LIN {X 0,Y 314.358,Z 529.66,A -85,B 0,C 180,E1 14023.753,E2 14023.753} C_VEL
LIN {X 0,Y 314.841,Z 529.66,A -85,B 0,C 180,E1 14031.737,E2 14031.737} C_VEL
LIN {X 0,Y 315.373,Z 529.66,A -85,B 0,C 180,E1 14037.261,E2 14037.261} C_VEL
LIN {X 0,Y 315.324,Z 529.66,A -85,B 0,C 180,E1 14042.747,E2 14042.747} C_VEL
LIN {X 0,Y 314.746,Z 529.66,A -85,B 0,C 180,E1 14051.06,E2 14051.06} C_VEL
LIN {X 0,Y 314.38,Z 529.66,A -85,B 0,C 180,E1 14056.741,E2 14056.741} C_VEL
LIN {X 0,Y 313.895,Z 529.66,A -85,B 0,C 180,E1 14064.019,E2 14064.019} C_VEL
LIN {X 0,Y 313.702,Z 529.66,A -85,B 0,C 180,E1 14072.529,E2 14072.529} C_VEL
LIN {X 0,Y 331.392,Z 572.539,A -85,B 0,C 180,E1 14075.795,E2 14075.795} C_VEL
LIN {X 0,Y 335.77,Z 585.842,A -85,B 0,C 180,E1 14076.583,E2 14076.583} C_VEL
LIN {X 0,Y 334.083,Z 636.564,A -85,B 0,C 180,E1 14077.88,E2 14077.88} C_VEL
LIN {X 0,Y 331.433,Z 665.303,A -85,B 0,C 180,E1 14079.603,E2 14079.603} C_VEL
LIN {X 0,Y 327.822,Z 690.981,A -85,B 0,C 180,E1 14082.214,E2 14082.214} C_VEL
LIN {X 0,Y 323.741,Z 713,A -85,B 0,C 180,E1 14085.638,E2 14085.638} C_VEL
LIN {X 0,Y 320.247,Z 730.569,A -85,B 0,C 180,E1 14089.741,E2 14089.741} C_VEL
LIN {X 0,Y 317.778,Z 743.68,A -85,B 0,C 180,E1 14094.497,E2 14094.497} C_VEL
LIN {X 0,Y 316.381,Z 751.07,A -85,B 0,C 180,E1 14099.156,E2 14099.156} C_VEL
LIN {X 0,Y 315.419,Z 754.016,A -85,B 0,C 180,E1 14104.495,E2 14104.495} C_VEL
LIN {X 0,Y 315.966,Z 751.687,A -85,B 0,C 180,E1 14109.434,E2 14109.434} C_VEL
LIN {X 0,Y 317.161,Z 744.828,A -85,B 0,C 180,E1 14114.122,E2 14114.122} C_VEL
LIN {X 0,Y 319.364,Z 731.71,A -85,B 0,C 180,E1 14119.104,E2 14119.104} C_VEL
LIN {X 0,Y 322.445,Z 714.366,A -85,B 0,C 180,E1 14123.28,E2 14123.28} C_VEL
LIN {X 0,Y 326.093,Z 692.368,A -85,B 0,C 180,E1 14126.826,E2 14126.826} C_VEL
LIN {X 0,Y 329.646,Z 666.051,A -85,B 0,C 180,E1 14129.589,E2 14129.589} C_VEL
LIN {X 0,Y 332.227,Z 637.274,A -85,B 0,C 180,E1 14131.367,E2 14131.367} C_VEL
LIN {X 0,Y 333.756,Z 589.127,A -85,B 0,C 180,E1 14132.637,E2 14132.637} C_VEL
LIN {X 0,Y 332.654,Z 578.727,A -85,B 0,C 180,E1 14132.982,E2 14132.982} C_VEL
LIN {X 0,Y 319.042,Z 540.423,A -85,B 0,C 180,E1 14135.188,E2 14135.188} C_VEL
LIN {X 0,Y 314.996,Z 529.66,A -85,B 0,C 180,E1 14136.014,E2 14136.014} C_VEL
LIN {X 0,Y 314.466,Z 529.66,A -85,B 0,C 180,E1 14143.881,E2 14143.881} C_VEL
LIN {X 0,Y 314.137,Z 529.66,A -85,B 0,C 180,E1 14149.647,E2 14149.647} C_VEL
LIN {X 0,Y 313.832,Z 529.66,A -85,B 0,C 180,E1 14155.641,E2 14155.641} C_VEL
LIN {X 0,Y 313.606,Z 529.66,A -85,B 0,C 180,E1 14161.956,E2 14161.956} C_VEL
LIN {X 0,Y 313.395,Z 529.66,A -85,B 0,C 180,E1 14169.605,E2 14169.605} C_VEL
LIN {X 0,Y 313.39,Z 529.66,A -85,B 0,C 180,E1 14177.611,E2 14177.611} C_VEL
LIN {X 0,Y 313.516,Z 529.661,A -85,B 0,C 180,E1 14178.724,E2 14178.724} C_VEL
LIN {X 0,Y 333.561,Z 579.091,A -85,B 0,C 180,E1 14182.875,E2 14182.875} C_VEL
LIN {X 0,Y 341.105,Z 602.01,A -85,B 0,C 180,E1 14185.002,E2 14185.002} C_VEL
LIN {X 0,Y 335.859,Z 636.992,A -85,B 0,C 180,E1 14187.695,E2 14187.695} C_VEL
LIN {X 0,Y 330.121,Z 668.653,A -85,B 0,C 180,E1 14191.314,E2 14191.314} C_VEL
LIN {X 0,Y 324.858,Z 695.392,A -85,B 0,C 180,E1 14195.65,E2 14195.65} C_VEL
LIN {X 0,Y 320.51,Z 717.686,A -85,B 0,C 180,E1 14200.754,E2 14200.754} C_VEL
LIN {X 0,Y 317.677,Z 734.305,A -85,B 0,C 180,E1 14206.257,E2 14206.257} C_VEL
LIN {X 0,Y 316.286,Z 745.604,A -85,B 0,C 180,E1 14212.1,E2 14212.1} C_VEL
LIN {X 0,Y 315.85,Z 751.035,A -85,B 0,C 180,E1 14217.258,E2 14217.258} C_VEL
LIN {X 0,Y 316.055,Z 752.334,A -85,B 0,C 180,E1 14222.733,E2 14222.733} C_VEL
LIN {X 0,Y 316.668,Z 749.149,A -85,B 0,C 180,E1 14228.215,E2 14228.215} C_VEL
LIN {X 0,Y 318.78,Z 740.37,A -85,B 0,C 180,E1 14234.24,E2 14234.24} C_VEL
LIN {X 0,Y 322.751,Z 725.649,A -85,B 0,C 180,E1 14240.202,E2 14240.202} C_VEL
LIN {X 0,Y 329.291,Z 704.647,A -85,B 0,C 180,E1 14245.803,E2 14245.803} C_VEL
LIN {X 0,Y 337.651,Z 677.968,A -85,B 0,C 180,E1 14250.736,E2 14250.736} C_VEL
LIN {X 0,Y 347.649,Z 645.626,A -85,B 0,C 180,E1 14254.914,E2 14254.914} C_VEL
LIN {X 0,Y 358.765,Z 606.435,A -85,B 0,C 180,E1 14258.535,E2 14258.535} C_VEL
LIN {X 0,Y 359.21,Z 596.015,A -85,B 0,C 180,E1 14260.875,E2 14260.875} C_VEL
LIN {X 0,Y 359.26,Z 593.944,A -85,B 0,C 180,E1 14262.22,E2 14262.22} C_VEL
LIN {X 0,Y 359.589,Z 594.189,A -85,B 0,C 180,E1 14263.651,E2 14263.651} C_VEL
LIN {X 0,Y 359.874,Z 599.525,A -85,B 0,C 180,E1 14265.46,E2 14265.46} C_VEL
LIN {X 0,Y 359.344,Z 611.481,A -85,B 0,C 180,E1 14267.298,E2 14267.298} C_VEL
LIN {X 0,Y 348.056,Z 653.394,A -85,B 0,C 180,E1 14270.652,E2 14270.652} C_VEL
LIN {X 0,Y 338.01,Z 689.08,A -85,B 0,C 180,E1 14274.803,E2 14274.803} C_VEL
LIN {X 0,Y 329.433,Z 719.409,A -85,B 0,C 180,E1 14279.745,E2 14279.745} C_VEL
LIN {X 0,Y 322.989,Z 743.295,A -85,B 0,C 180,E1 14285.137,E2 14285.137} C_VEL
LIN {X 0,Y 318.517,Z 762.82,A -85,B 0,C 180,E1 14291.34,E2 14291.34} C_VEL
LIN {X 0,Y 316.479,Z 775.559,A -85,B 0,C 180,E1 14297.373,E2 14297.373} C_VEL
LIN {X 0,Y 315.859,Z 782.903,A -85,B 0,C 180,E1 14303.142,E2 14303.142} C_VEL
LIN {X 0,Y 315.765,Z 785.334,A -85,B 0,C 180,E1 14307.262,E2 14307.262} C_VEL
LIN {X 0,Y 315.855,Z 784.953,A -85,B 0,C 180,E1 14312.74,E2 14312.74} C_VEL
LIN {X 0,Y 315.941,Z 780.256,A -85,B 0,C 180,E1 14318.239,E2 14318.239} C_VEL
LIN {X 0,Y 316.897,Z 769.663,A -85,B 0,C 180,E1 14324.478,E2 14324.478} C_VEL
LIN {X 0,Y 319.276,Z 753.654,A -85,B 0,C 180,E1 14330.401,E2 14330.401} C_VEL
LIN {X 0,Y 323.428,Z 732.194,A -85,B 0,C 180,E1 14335.939,E2 14335.939} C_VEL
LIN {X 0,Y 325.518,Z 722.568,A -85,B 0,C 180,E1 14337.919,E2 14337.919} C_VEL
LIN {X 0,Y 324.253,Z 710.874,A -85,B 0,C 180,E1 14340.211,E2 14340.211} C_VEL
LIN {X 0,Y 323.099,Z 698.429,A -85,B 0,C 180,E1 14342.396,E2 14342.396} C_VEL
LIN {X 0,Y 329.898,Z 665.459,A -85,B 0,C 180,E1 14346.488,E2 14346.488} C_VEL
LIN {X 0,Y 336.27,Z 629.393,A -85,B 0,C 180,E1 14349.577,E2 14349.577} C_VEL
LIN {X 0,Y 338.64,Z 610.74,A -85,B 0,C 180,E1 14350.76,E2 14350.76} C_VEL
LIN {X 0,Y 324.137,Z 572.197,A -85,B 0,C 180,E1 14354.249,E2 14354.249} C_VEL
LIN {X 0,Y 305.579,Z 529.66,A -85,B 0,C 180,E1 14358.2,E2 14358.2} C_VEL
LIN {X 0,Y 305.614,Z 529.66,A -85,B 0,C 180,E1 14367.108,E2 14367.108} C_VEL
LIN {X 0,Y 305.857,Z 529.66,A -85,B 0,C 180,E1 14373.643,E2 14373.643} C_VEL
LIN {X 0,Y 306.152,Z 529.66,A -85,B 0,C 180,E1 14379.821,E2 14379.821} C_VEL
LIN {X 0,Y 306.519,Z 529.66,A -85,B 0,C 180,E1 14385.754,E2 14385.754} C_VEL
LIN {X 0,Y 306.894,Z 529.66,A -85,B 0,C 180,E1 14391.521,E2 14391.521} C_VEL
LIN {X 0,Y 307.45,Z 529.66,A -85,B 0,C 180,E1 14397.191,E2 14397.191} C_VEL
LIN {X 0,Y 307.404,Z 529.66,A -85,B 0,C 180,E1 14402.817,E2 14402.817} C_VEL
LIN {X 0,Y 306.811,Z 529.66,A -85,B 0,C 180,E1 14411.35,E2 14411.35} C_VEL
LIN {X 0,Y 306.396,Z 529.66,A -85,B 0,C 180,E1 14417.191,E2 14417.191} C_VEL
LIN {X 0,Y 306.041,Z 529.66,A -85,B 0,C 180,E1 14423.236,E2 14423.236} C_VEL
LIN {X 0,Y 305.753,Z 529.66,A -85,B 0,C 180,E1 14431.48,E2 14431.48} C_VEL
LIN {X 0,Y 323.99,Z 572.634,A -85,B 0,C 180,E1 14434.995,E2 14434.995} C_VEL
LIN {X 0,Y 328.959,Z 588.44,A -85,B 0,C 180,E1 14435.949,E2 14435.949} C_VEL
LIN {X 0,Y 327.127,Z 637.889,A -85,B 0,C 180,E1 14437.26,E2 14437.26} C_VEL
LIN {X 0,Y 324.455,Z 665.524,A -85,B 0,C 180,E1 14438.961,E2 14438.961} C_VEL
LIN {X 0,Y 320.62,Z 691.541,A -85,B 0,C 180,E1 14441.656,E2 14441.656} C_VEL
LIN {X 0,Y 316.272,Z 713.758,A -85,B 0,C 180,E1 14445.199,E2 14445.199} C_VEL
LIN {X 0,Y 312.4,Z 732.228,A -85,B 0,C 180,E1 14449.7,E2 14449.7} C_VEL
LIN {X 0,Y 309.987,Z 744.201,A -85,B 0,C 180,E1 14454.256,E2 14454.256} C_VEL
LIN {X 0,Y 308.375,Z 752.077,A -85,B 0,C 180,E1 14459.556,E2 14459.556} C_VEL
LIN {X 0,Y 307.546,Z 754.341,A -85,B 0,C 180,E1 14463.793,E2 14463.793} C_VEL
LIN {X 0,Y 307.872,Z 752.827,A -85,B 0,C 180,E1 14468.64,E2 14468.64} C_VEL
LIN {X 0,Y 309.126,Z 746.371,A -85,B 0,C 180,E1 14473.698,E2 14473.698} C_VEL
LIN {X 0,Y 311.331,Z 733.969,A -85,B 0,C 180,E1 14478.82,E2 14478.82} C_VEL
LIN {X 0,Y 314.366,Z 717.563,A -85,B 0,C 180,E1 14483.107,E2 14483.107} C_VEL
LIN {X 0,Y 318.132,Z 696.355,A -85,B 0,C 180,E1 14486.818,E2 14486.818} C_VEL
LIN {X 0,Y 321.802,Z 671.686,A -85,B 0,C 180,E1 14489.663,E2 14489.663} C_VEL
LIN {X 0,Y 324.629,Z 643.608,A -85,B 0,C 180,E1 14491.662,E2 14491.662} C_VEL
LIN {X 0,Y 326.15,Z 611.366,A -85,B 0,C 180,E1 14492.747,E2 14492.747} C_VEL
LIN {X 0,Y 326.263,Z 582.825,A -85,B 0,C 180,E1 14493.443,E2 14493.443} C_VEL
LIN {X 0,Y 312.895,Z 544.522,A -85,B 0,C 180,E1 14495.694,E2 14495.694} C_VEL
LIN {X 0,Y 307.04,Z 529.66,A -85,B 0,C 180,E1 14496.791,E2 14496.791} C_VEL
LIN {X 0,Y 306.534,Z 529.66,A -85,B 0,C 180,E1 14504.248,E2 14504.248} C_VEL
LIN {X 0,Y 306.028,Z 529.66,A -85,B 0,C 180,E1 14513.232,E2 14513.232} C_VEL
LIN {X 0,Y 305.731,Z 529.66,A -85,B 0,C 180,E1 14519.574,E2 14519.574} C_VEL
LIN {X 0,Y 305.424,Z 529.66,A -85,B 0,C 180,E1 14527.762,E2 14527.762} C_VEL
LIN {X 0,Y 305.501,Z 529.66,A -85,B 0,C 180,E1 14533.748,E2 14533.748} C_VEL
LIN {X 0,Y 305.523,Z 529.888,A -85,B 0,C 180,E1 14537.803,E2 14537.803} C_VEL
LIN {X 0,Y 325.664,Z 578.93,A -85,B 0,C 180,E1 14542.105,E2 14542.105} C_VEL
LIN {X 0,Y 333.718,Z 604.557,A -85,B 0,C 180,E1 14544.541,E2 14544.541} C_VEL
LIN {X 0,Y 328.331,Z 638.995,A -85,B 0,C 180,E1 14547.311,E2 14547.311} C_VEL
LIN {X 0,Y 322.326,Z 670.994,A -85,B 0,C 180,E1 14551.129,E2 14551.129} C_VEL
LIN {X 0,Y 316.772,Z 698.028,A -85,B 0,C 180,E1 14555.737,E2 14555.737} C_VEL
LIN {X 0,Y 312.44,Z 719.749,A -85,B 0,C 180,E1 14560.97,E2 14560.97} C_VEL
LIN {X 0,Y 309.608,Z 736.118,A -85,B 0,C 180,E1 14566.718,E2 14566.718} C_VEL
LIN {X 0,Y 308.409,Z 745.967,A -85,B 0,C 180,E1 14572.065,E2 14572.065} C_VEL
LIN {X 0,Y 307.959,Z 751.348,A -85,B 0,C 180,E1 14577.188,E2 14577.188} C_VEL
LIN {X 0,Y 308.171,Z 752.848,A -85,B 0,C 180,E1 14582.803,E2 14582.803} C_VEL
LIN {X 0,Y 308.884,Z 749.882,A -85,B 0,C 180,E1 14588.424,E2 14588.424} C_VEL
LIN {X 0,Y 311.217,Z 741.069,A -85,B 0,C 180,E1 14594.743,E2 14594.743} C_VEL
LIN {X 0,Y 315.609,Z 726.484,A -85,B 0,C 180,E1 14600.863,E2 14600.863} C_VEL
LIN {X 0,Y 322.412,Z 706.547,A -85,B 0,C 180,E1 14606.395,E2 14606.395} C_VEL
LIN {X 0,Y 331.615,Z 679.844,A -85,B 0,C 180,E1 14611.549,E2 14611.549} C_VEL
LIN {X 0,Y 342.737,Z 647.661,A -85,B 0,C 180,E1 14615.877,E2 14615.877} C_VEL
LIN {X 0,Y 354.943,Z 610.837,A -85,B 0,C 180,E1 14619.396,E2 14619.396} C_VEL
LIN {X 0,Y 356.118,Z 602.755,A -85,B 0,C 180,E1 14621.307,E2 14621.307} C_VEL
LIN {X 0,Y 356.354,Z 601.212,A -85,B 0,C 180,E1 14622.645,E2 14622.645} C_VEL
LIN {X 0,Y 356.581,Z 602.503,A -85,B 0,C 180,E1 14623.996,E2 14623.996} C_VEL
LIN {X 0,Y 355.793,Z 610.922,A -85,B 0,C 180,E1 14625.831,E2 14625.831} C_VEL
LIN {X 0,Y 353.664,Z 619.82,A -85,B 0,C 180,E1 14626.696,E2 14626.696} C_VEL
LIN {X 0,Y 341.465,Z 659.253,A -85,B 0,C 180,E1 14630.151,E2 14630.151} C_VEL
LIN {X 0,Y 330.11,Z 695.501,A -85,B 0,C 180,E1 14634.755,E2 14634.755} C_VEL
LIN {X 0,Y 321.145,Z 724.9,A -85,B 0,C 180,E1 14640.03,E2 14640.03} C_VEL
LIN {X 0,Y 314.432,Z 748.303,A -85,B 0,C 180,E1 14645.916,E2 14645.916} C_VEL
LIN {X 0,Y 310.069,Z 766.678,A -85,B 0,C 180,E1 14652.533,E2 14652.533} C_VEL
LIN {X 0,Y 308.382,Z 777.819,A -85,B 0,C 180,E1 14658.714,E2 14658.714} C_VEL
LIN {X 0,Y 307.923,Z 783.588,A -85,B 0,C 180,E1 14664.377,E2 14664.377} C_VEL
LIN {X 0,Y 308.005,Z 785.155,A -85,B 0,C 180,E1 14670.001,E2 14670.001} C_VEL
LIN {X 0,Y 307.938,Z 782.501,A -85,B 0,C 180,E1 14675.626,E2 14675.626} C_VEL
LIN {X 0,Y 308.489,Z 774.306,A -85,B 0,C 180,E1 14681.976,E2 14681.976} C_VEL
LIN {X 0,Y 310.305,Z 760.118,A -85,B 0,C 180,E1 14688.366,E2 14688.366} C_VEL
LIN {X 0,Y 313.903,Z 740.758,A -85,B 0,C 180,E1 14694.194,E2 14694.194} C_VEL
LIN {X 0,Y 319.199,Z 716.347,A -85,B 0,C 180,E1 14699.442,E2 14699.442} C_VEL
LIN {X 0,Y 323.099,Z 698.429,A -85,B 0,C 180,E1 14702.396,E2 14702.396} C_VEL
LIN {X 0,Y 322.145,Z 685.268,A -85,B 0,C 180,E1 14704.454,E2 14704.454} C_VEL
LIN {X 0,Y 321.126,Z 673.313,A -85,B 0,C 180,E1 14706.165,E2 14706.165} C_VEL
LIN {X 0,Y 321.449,Z 671.49,A -85,B 0,C 180,E1 14706.381,E2 14706.381} C_VEL
LIN {X 0,Y 328.131,Z 636.403,A -85,B 0,C 180,E1 14709.66,E2 14709.66} C_VEL
LIN {X 0,Y 331.334,Z 612.5,A -85,B 0,C 180,E1 14711.302,E2 14711.302} C_VEL
LIN {X 0,Y 317.076,Z 574.226,A -85,B 0,C 180,E1 14714.919,E2 14714.919} C_VEL
LIN {X 0,Y 297.595,Z 529.66,A -85,B 0,C 180,E1 14719.2,E2 14719.2} C_VEL
LIN {X 0,Y 297.585,Z 529.66,A -85,B 0,C 180,E1 14726.102,E2 14726.102} C_VEL
LIN {X 0,Y 297.887,Z 529.66,A -85,B 0,C 180,E1 14732.881,E2 14732.881} C_VEL
LIN {X 0,Y 298.194,Z 529.66,A -85,B 0,C 180,E1 14739.258,E2 14739.258} C_VEL
LIN {X 0,Y 298.542,Z 529.66,A -85,B 0,C 180,E1 14745.365,E2 14745.365} C_VEL
LIN {X 0,Y 299.193,Z 529.66,A -85,B 0,C 180,E1 14754.215,E2 14754.215} C_VEL
LIN {X 0,Y 299.684,Z 529.66,A -85,B 0,C 180,E1 14760.004,E2 14760.004} C_VEL
LIN {X 0,Y 299.216,Z 529.66,A -85,B 0,C 180,E1 14765.793,E2 14765.793} C_VEL
LIN {X 0,Y 298.848,Z 529.66,A -85,B 0,C 180,E1 14771.656,E2 14771.656} C_VEL
LIN {X 0,Y 298.427,Z 529.66,A -85,B 0,C 180,E1 14777.665,E2 14777.665} C_VEL
LIN {X 0,Y 297.966,Z 529.66,A -85,B 0,C 180,E1 14784.273,E2 14784.273} C_VEL
LIN {X 0,Y 297.813,Z 529.66,A -85,B 0,C 180,E1 14790.301,E2 14790.301} C_VEL
LIN {X 0,Y 315.69,Z 570.347,A -85,B 0,C 180,E1 14793.97,E2 14793.97} C_VEL
LIN {X 0,Y 322.179,Z 589.324,A -85,B 0,C 180,E1 14795.239,E2 14795.239} C_VEL
LIN {X 0,Y 320.281,Z 638.358,A -85,B 0,C 180,E1 14796.569,E2 14796.569} C_VEL
LIN {X 0,Y 317.266,Z 667.514,A -85,B 0,C 180,E1 14798.425,E2 14798.425} C_VEL
LIN {X 0,Y 313.164,Z 693.514,A -85,B 0,C 180,E1 14801.256,E2 14801.256} C_VEL
LIN {X 0,Y 308.621,Z 715.606,A -85,B 0,C 180,E1 14804.966,E2 14804.966} C_VEL
LIN {X 0,Y 304.774,Z 732.841,A -85,B 0,C 180,E1 14809.334,E2 14809.334} C_VEL
LIN {X 0,Y 302.154,Z 745.012,A -85,B 0,C 180,E1 14814.135,E2 14814.135} C_VEL
LIN {X 0,Y 300.753,Z 751.612,A -85,B 0,C 180,E1 14818.541,E2 14818.541} C_VEL
LIN {X 0,Y 299.725,Z 754.61,A -85,B 0,C 180,E1 14823.055,E2 14823.055} C_VEL
LIN {X 0,Y 299.626,Z 754.512,A -85,B 0,C 180,E1 14826.239,E2 14826.239} C_VEL
LIN {X 0,Y 300.504,Z 751.038,A -85,B 0,C 180,E1 14830.95,E2 14830.95} C_VEL
LIN {X 0,Y 302.234,Z 741.471,A -85,B 0,C 180,E1 14836.471,E2 14836.471} C_VEL
LIN {X 0,Y 305.134,Z 726.208,A -85,B 0,C 180,E1 14841.541,E2 14841.541} C_VEL
LIN {X 0,Y 308.926,Z 706.357,A -85,B 0,C 180,E1 14845.783,E2 14845.783} C_VEL
LIN {X 0,Y 313.033,Z 682.517,A -85,B 0,C 180,E1 14849.136,E2 14849.136} C_VEL
LIN {X 0,Y 316.449,Z 655.272,A -85,B 0,C 180,E1 14851.581,E2 14851.581} C_VEL
LIN {X 0,Y 318.626,Z 625.599,A -85,B 0,C 180,E1 14853.013,E2 14853.013} C_VEL
LIN {X 0,Y 319.224,Z 584.419,A -85,B 0,C 180,E1 14854.041,E2 14854.041} C_VEL
LIN {X 0,Y 305.58,Z 545.612,A -85,B 0,C 180,E1 14856.427,E2 14856.427} C_VEL
LIN {X 0,Y 299.053,Z 529.66,A -85,B 0,C 180,E1 14857.651,E2 14857.651} C_VEL
LIN {X 0,Y 298.433,Z 529.66,A -85,B 0,C 180,E1 14866.103,E2 14866.103} C_VEL
LIN {X 0,Y 297.955,Z 529.66,A -85,B 0,C 180,E1 14874.264,E2 14874.264} C_VEL
LIN {X 0,Y 297.706,Z 529.66,A -85,B 0,C 180,E1 14880.487,E2 14880.487} C_VEL
LIN {X 0,Y 297.52,Z 529.66,A -85,B 0,C 180,E1 14887.489,E2 14887.489} C_VEL
LIN {X 0,Y 297.553,Z 529.66,A -85,B 0,C 180,E1 14895.232,E2 14895.232} C_VEL
LIN {X 0,Y 297.613,Z 530.095,A -85,B 0,C 180,E1 14896.853,E2 14896.853} C_VEL
LIN {X 0,Y 318.04,Z 579.56,A -85,B 0,C 180,E1 14901.388,E2 14901.388} C_VEL
LIN {X 0,Y 326.532,Z 605.74,A -85,B 0,C 180,E1 14903.995,E2 14903.995} C_VEL
LIN {X 0,Y 320.907,Z 640.317,A -85,B 0,C 180,E1 14906.86,E2 14906.86} C_VEL
LIN {X 0,Y 314.682,Z 672.215,A -85,B 0,C 180,E1 14910.783,E2 14910.783} C_VEL
LIN {X 0,Y 309.062,Z 698.904,A -85,B 0,C 180,E1 14915.476,E2 14915.476} C_VEL
LIN {X 0,Y 304.537,Z 720.848,A -85,B 0,C 180,E1 14920.94,E2 14920.94} C_VEL
LIN {X 0,Y 301.667,Z 737.138,A -85,B 0,C 180,E1 14926.869,E2 14926.869} C_VEL
LIN {X 0,Y 300.46,Z 747.384,A -85,B 0,C 180,E1 14932.783,E2 14932.783} C_VEL
LIN {X 0,Y 300.067,Z 751.649,A -85,B 0,C 180,E1 14937.114,E2 14937.114} C_VEL
LIN {X 0,Y 300.286,Z 753.349,A -85,B 0,C 180,E1 14942.877,E2 14942.877} C_VEL
LIN {X 0,Y 301.072,Z 750.61,A -85,B 0,C 180,E1 14948.644,E2 14948.644} C_VEL
LIN {X 0,Y 303.604,Z 742.099,A -85,B 0,C 180,E1 14955.122,E2 14955.122} C_VEL
LIN {X 0,Y 308.262,Z 728.195,A -85,B 0,C 180,E1 14961.293,E2 14961.293} C_VEL
LIN {X 0,Y 316.045,Z 707.518,A -85,B 0,C 180,E1 14967.262,E2 14967.262} C_VEL
LIN {X 0,Y 326.097,Z 681.087,A -85,B 0,C 180,E1 14972.539,E2 14972.539} C_VEL
LIN {X 0,Y 338.508,Z 649.013,A -85,B 0,C 180,E1 14976.994,E2 14976.994} C_VEL
LIN {X 0,Y 351.568,Z 614.752,A -85,B 0,C 180,E1 14980.392,E2 14980.392} C_VEL
LIN {X 0,Y 352.913,Z 609.452,A -85,B 0,C 180,E1 14981.841,E2 14981.841} C_VEL
LIN {X 0,Y 353.236,Z 609.749,A -85,B 0,C 180,E1 14983.727,E2 14983.727} C_VEL
LIN {X 0,Y 351.588,Z 617.781,A -85,B 0,C 180,E1 14985.29,E2 14985.29} C_VEL
LIN {X 0,Y 337.23,Z 658.601,A -85,B 0,C 180,E1 14988.915,E2 14988.915} C_VEL
LIN {X 0,Y 324.541,Z 695.001,A -85,B 0,C 180,E1 14993.644,E2 14993.644} C_VEL
LIN {X 0,Y 314.521,Z 724.816,A -85,B 0,C 180,E1 14999.142,E2 14999.142} C_VEL
LIN {X 0,Y 307.071,Z 748.519,A -85,B 0,C 180,E1 15005.301,E2 15005.301} C_VEL
LIN {X 0,Y 302.448,Z 766.205,A -85,B 0,C 180,E1 15011.899,E2 15011.899} C_VEL
LIN {X 0,Y 300.527,Z 777.54,A -85,B 0,C 180,E1 15018.415,E2 15018.415} C_VEL
LIN {X 0,Y 300.056,Z 783.229,A -85,B 0,C 180,E1 15024.229,E2 15024.229} C_VEL
LIN {X 0,Y 300.145,Z 784.668,A -85,B 0,C 180,E1 15030.001,E2 15030.001} C_VEL
LIN {X 0,Y 300.069,Z 781.86,A -85,B 0,C 180,E1 15035.774,E2 15035.774} C_VEL
LIN {X 0,Y 300.558,Z 774.646,A -85,B 0,C 180,E1 15041.586,E2 15041.586} C_VEL
LIN {X 0,Y 302.27,Z 761.115,A -85,B 0,C 180,E1 15048.031,E2 15048.031} C_VEL
LIN {X 0,Y 305.994,Z 741.396,A -85,B 0,C 180,E1 15054.273,E2 15054.273} C_VEL
LIN {X 0,Y 311.358,Z 717.32,A -85,B 0,C 180,E1 15059.636,E2 15059.636} C_VEL
LIN {X 0,Y 318.129,Z 687.037,A -85,B 0,C 180,E1 15064.469,E2 15064.469} C_VEL
LIN {X 0,Y 321.449,Z 671.49,A -85,B 0,C 180,E1 15066.381,E2 15066.381} C_VEL
LIN {X 0,Y 320.746,Z 657.119,A -85,B 0,C 180,E1 15068.167,E2 15068.167} C_VEL
LIN {X 0,Y 319.707,Z 644.164,A -85,B 0,C 180,E1 15069.633,E2 15069.633} C_VEL
LIN {X 0,Y 320.014,Z 642.199,A -85,B 0,C 180,E1 15069.807,E2 15069.807} C_VEL
LIN {X 0,Y 324.059,Z 614.344,A -85,B 0,C 180,E1 15071.843,E2 15071.843} C_VEL
LIN {X 0,Y 309.999,Z 576.256,A -85,B 0,C 180,E1 15075.6,E2 15075.6} C_VEL
LIN {X 0,Y 289.601,Z 529.66,A -85,B 0,C 180,E1 15080.182,E2 15080.182} C_VEL
LIN {X 0,Y 289.701,Z 529.66,A -85,B 0,C 180,E1 15088.614,E2 15088.614} C_VEL
LIN {X 0,Y 290.033,Z 529.66,A -85,B 0,C 180,E1 15095.408,E2 15095.408} C_VEL
LIN {X 0,Y 290.37,Z 529.66,A -85,B 0,C 180,E1 15101.836,E2 15101.836} C_VEL
LIN {X 0,Y 290.909,Z 529.66,A -85,B 0,C 180,E1 15110.258,E2 15110.258} C_VEL
LIN {X 0,Y 291.626,Z 529.66,A -85,B 0,C 180,E1 15117.038,E2 15117.038} C_VEL
LIN {X 0,Y 291.573,Z 529.66,A -85,B 0,C 180,E1 15122.971,E2 15122.971} C_VEL
LIN {X 0,Y 290.888,Z 529.66,A -85,B 0,C 180,E1 15131.98,E2 15131.98} C_VEL
LIN {X 0,Y 290.334,Z 529.66,A -85,B 0,C 180,E1 15140.681,E2 15140.681} C_VEL
LIN {X 0,Y 289.94,Z 529.66,A -85,B 0,C 180,E1 15149.088,E2 15149.088} C_VEL
LIN {X 0,Y 308.195,Z 570.236,A -85,B 0,C 180,E1 15153.033,E2 15153.033} C_VEL
LIN {X 0,Y 315.448,Z 592.213,A -85,B 0,C 180,E1 15154.547,E2 15154.547} C_VEL
LIN {X 0,Y 313.436,Z 639.479,A -85,B 0,C 180,E1 15155.876,E2 15155.876} C_VEL
LIN {X 0,Y 310.311,Z 668.206,A -85,B 0,C 180,E1 15157.759,E2 15157.759} C_VEL
LIN {X 0,Y 306.013,Z 694.13,A -85,B 0,C 180,E1 15160.649,E2 15160.649} C_VEL
LIN {X 0,Y 301.119,Z 716.738,A -85,B 0,C 180,E1 15164.558,E2 15164.558} C_VEL
LIN {X 0,Y 296.898,Z 734.541,A -85,B 0,C 180,E1 15169.303,E2 15169.303} C_VEL
LIN {X 0,Y 294.126,Z 746.78,A -85,B 0,C 180,E1 15174.565,E2 15174.565} C_VEL
LIN {X 0,Y 292.751,Z 752.66,A -85,B 0,C 180,E1 15178.971,E2 15178.971} C_VEL
LIN {X 0,Y 291.918,Z 754.782,A -85,B 0,C 180,E1 15182.273,E2 15182.273} C_VEL
LIN {X 0,Y 291.722,Z 755.063,A -85,B 0,C 180,E1 15185.554,E2 15185.554} C_VEL
LIN {X 0,Y 292.457,Z 752.118,A -85,B 0,C 180,E1 15190.403,E2 15190.403} C_VEL
LIN {X 0,Y 294.018,Z 744.185,A -85,B 0,C 180,E1 15195.638,E2 15195.638} C_VEL
LIN {X 0,Y 296.711,Z 730.356,A -85,B 0,C 180,E1 15200.854,E2 15200.854} C_VEL
LIN {X 0,Y 300.463,Z 711.814,A -85,B 0,C 180,E1 15205.319,E2 15205.319} C_VEL
LIN {X 0,Y 304.945,Z 687.701,A -85,B 0,C 180,E1 15209.113,E2 15209.113} C_VEL
LIN {X 0,Y 308.664,Z 661.187,A -85,B 0,C 180,E1 15211.778,E2 15211.778} C_VEL
LIN {X 0,Y 311.274,Z 631.423,A -85,B 0,C 180,E1 15213.461,E2 15213.461} C_VEL
LIN {X 0,Y 312.143,Z 585.984,A -85,B 0,C 180,E1 15214.674,E2 15214.674} C_VEL
LIN {X 0,Y 299.148,Z 548.955,A -85,B 0,C 180,E1 15217.029,E2 15217.029} C_VEL
LIN {X 0,Y 291.103,Z 529.66,A -85,B 0,C 180,E1 15218.669,E2 15218.669} C_VEL
LIN {X 0,Y 290.601,Z 529.66,A -85,B 0,C 180,E1 15225.047,E2 15225.047} C_VEL
LIN {X 0,Y 290.201,Z 529.66,A -85,B 0,C 180,E1 15231.344,E2 15231.344} C_VEL
LIN {X 0,Y 289.83,Z 529.66,A -85,B 0,C 180,E1 15237.941,E2 15237.941} C_VEL
LIN {X 0,Y 289.619,Z 529.66,A -85,B 0,C 180,E1 15244.967,E2 15244.967} C_VEL
LIN {X 0,Y 289.49,Z 529.66,A -85,B 0,C 180,E1 15253.129,E2 15253.129} C_VEL
LIN {X 0,Y 289.692,Z 530.377,A -85,B 0,C 180,E1 15255.868,E2 15255.868} C_VEL
LIN {X 0,Y 310.037,Z 579.233,A -85,B 0,C 180,E1 15260.55,E2 15260.55} C_VEL
LIN {X 0,Y 319.308,Z 607.182,A -85,B 0,C 180,E1 15263.453,E2 15263.453} C_VEL
LIN {X 0,Y 313.515,Z 641.457,A -85,B 0,C 180,E1 15266.388,E2 15266.388} C_VEL
LIN {X 0,Y 307.12,Z 673.133,A -85,B 0,C 180,E1 15270.392,E2 15270.392} C_VEL
LIN {X 0,Y 301.185,Z 700.315,A -85,B 0,C 180,E1 15275.327,E2 15275.327} C_VEL
LIN {X 0,Y 296.603,Z 721.922,A -85,B 0,C 180,E1 15280.914,E2 15280.914} C_VEL
LIN {X 0,Y 293.897,Z 737.002,A -85,B 0,C 180,E1 15286.531,E2 15286.531} C_VEL
LIN {X 0,Y 292.597,Z 747.522,A -85,B 0,C 180,E1 15292.588,E2 15292.588} C_VEL
LIN {X 0,Y 292.176,Z 751.939,A -85,B 0,C 180,E1 15297.036,E2 15297.036} C_VEL
LIN {X 0,Y 292.402,Z 753.854,A -85,B 0,C 180,E1 15302.954,E2 15302.954} C_VEL
LIN {X 0,Y 293.295,Z 751.339,A -85,B 0,C 180,E1 15308.875,E2 15308.875} C_VEL
LIN {X 0,Y 296.028,Z 743.186,A -85,B 0,C 180,E1 15315.518,E2 15315.518} C_VEL
LIN {X 0,Y 301.055,Z 729.685,A -85,B 0,C 180,E1 15321.829,E2 15321.829} C_VEL
LIN {X 0,Y 309.48,Z 709.388,A -85,B 0,C 180,E1 15327.985,E2 15327.985} C_VEL
LIN {X 0,Y 320.778,Z 682.68,A -85,B 0,C 180,E1 15333.55,E2 15333.55} C_VEL
LIN {X 0,Y 334.591,Z 651.002,A -85,B 0,C 180,E1 15338.114,E2 15338.114} C_VEL
LIN {X 0,Y 348.585,Z 619.222,A -85,B 0,C 180,E1 15341.361,E2 15341.361} C_VEL
LIN {X 0,Y 349.246,Z 617.417,A -85,B 0,C 180,E1 15341.821,E2 15341.821} C_VEL
LIN {X 0,Y 349.808,Z 616.232,A -85,B 0,C 180,E1 15342.834,E2 15342.834} C_VEL
LIN {X 0,Y 348.956,Z 619.544,A -85,B 0,C 180,E1 15343.982,E2 15343.982} C_VEL
LIN {X 0,Y 330.857,Z 664.932,A -85,B 0,C 180,E1 15348.383,E2 15348.383} C_VEL
LIN {X 0,Y 316.935,Z 700.81,A -85,B 0,C 180,E1 15353.48,E2 15353.48} C_VEL
LIN {X 0,Y 306.39,Z 729.375,A -85,B 0,C 180,E1 15359.246,E2 15359.246} C_VEL
LIN {X 0,Y 298.777,Z 752.132,A -85,B 0,C 180,E1 15365.775,E2 15365.775} C_VEL
LIN {X 0,Y 294.131,Z 769.011,A -85,B 0,C 180,E1 15372.844,E2 15372.844} C_VEL
LIN {X 0,Y 292.436,Z 779.27,A -85,B 0,C 180,E1 15379.761,E2 15379.761} C_VEL
LIN {X 0,Y 292.157,Z 782.84,A -85,B 0,C 180,E1 15384.072,E2 15384.072} C_VEL
LIN {X 0,Y 292.256,Z 784.176,A -85,B 0,C 180,E1 15390.001,E2 15390.001} C_VEL
LIN {X 0,Y 292.18,Z 781.199,A -85,B 0,C 180,E1 15395.93,E2 15395.93} C_VEL
LIN {X 0,Y 292.702,Z 773.778,A -85,B 0,C 180,E1 15401.902,E2 15401.902} C_VEL
LIN {X 0,Y 294.548,Z 759.985,A -85,B 0,C 180,E1 15408.52,E2 15408.52} C_VEL
LIN {X 0,Y 298.353,Z 740.572,A -85,B 0,C 180,E1 15414.725,E2 15414.725} C_VEL
LIN {X 0,Y 303.918,Z 716.471,A -85,B 0,C 180,E1 15420.181,E2 15420.181} C_VEL
LIN {X 0,Y 310.908,Z 686.177,A -85,B 0,C 180,E1 15425.082,E2 15425.082} C_VEL
LIN {X 0,Y 318.062,Z 652.008,A -85,B 0,C 180,E1 15428.95,E2 15428.95} C_VEL
LIN {X 0,Y 320.014,Z 642.199,A -85,B 0,C 180,E1 15429.807,E2 15429.807} C_VEL
LIN {X 0,Y 320.241,Z 630.497,A -85,B 0,C 180,E1 15430.895,E2 15430.895} C_VEL
LIN {X 0,Y 315.274,Z 611.7,A -85,B 0,C 180,E1 15432.885,E2 15432.885} C_VEL
LIN {X 0,Y 301.436,Z 574.781,A -85,B 0,C 180,E1 15436.632,E2 15436.632} C_VEL
LIN {X 0,Y 281.695,Z 529.66,A -85,B 0,C 180,E1 15441.194,E2 15441.194} C_VEL
LIN {X 0,Y 281.771,Z 529.66,A -85,B 0,C 180,E1 15448.969,E2 15448.969} C_VEL
LIN {X 0,Y 282.14,Z 529.66,A -85,B 0,C 180,E1 15455.401,E2 15455.401} C_VEL
LIN {X 0,Y 282.602,Z 529.66,A -85,B 0,C 180,E1 15464.52,E2 15464.52} C_VEL
LIN {X 0,Y 283.076,Z 529.66,A -85,B 0,C 180,E1 15470.802,E2 15470.802} C_VEL
LIN {X 0,Y 283.696,Z 529.66,A -85,B 0,C 180,E1 15476.955,E2 15476.955} C_VEL
LIN {X 0,Y 283.648,Z 529.66,A -85,B 0,C 180,E1 15483.054,E2 15483.054} C_VEL
LIN {X 0,Y 282.919,Z 529.66,A -85,B 0,C 180,E1 15492.323,E2 15492.323} C_VEL
LIN {X 0,Y 282.465,Z 529.66,A -85,B 0,C 180,E1 15498.699,E2 15498.699} C_VEL
LIN {X 0,Y 282.039,Z 529.66,A -85,B 0,C 180,E1 15507.725,E2 15507.725} C_VEL
LIN {X 0,Y 289.194,Z 544.62,A -85,B 0,C 180,E1 15509.505,E2 15509.505} C_VEL
LIN {X 0,Y 303.919,Z 578.379,A -85,B 0,C 180,E1 15512.711,E2 15512.711} C_VEL
LIN {X 0,Y 308.77,Z 594.917,A -85,B 0,C 180,E1 15513.816,E2 15513.816} C_VEL
LIN {X 0,Y 306.75,Z 639.663,A -85,B 0,C 180,E1 15515.102,E2 15515.102} C_VEL
LIN {X 0,Y 303.371,Z 669.165,A -85,B 0,C 180,E1 15517.075,E2 15517.075} C_VEL
LIN {X 0,Y 298.836,Z 695.035,A -85,B 0,C 180,E1 15520.05,E2 15520.05} C_VEL
LIN {X 0,Y 293.754,Z 717.327,A -85,B 0,C 180,E1 15524.012,E2 15524.012} C_VEL
LIN {X 0,Y 289.432,Z 734.586,A -85,B 0,C 180,E1 15528.702,E2 15528.702} C_VEL
LIN {X 0,Y 286.399,Z 747.104,A -85,B 0,C 180,E1 15534.185,E2 15534.185} C_VEL
LIN {X 0,Y 284.752,Z 753.532,A -85,B 0,C 180,E1 15539.326,E2 15539.326} C_VEL
LIN {X 0,Y 283.803,Z 755.545,A -85,B 0,C 180,E1 15544.825,E2 15544.825} C_VEL
LIN {X 0,Y 284.423,Z 753.157,A -85,B 0,C 180,E1 15549.826,E2 15549.826} C_VEL
LIN {X 0,Y 286.096,Z 745.197,A -85,B 0,C 180,E1 15555.564,E2 15555.564} C_VEL
LIN {X 0,Y 288.879,Z 731.514,A -85,B 0,C 180,E1 15560.983,E2 15560.983} C_VEL
LIN {X 0,Y 292.745,Z 713.374,A -85,B 0,C 180,E1 15565.564,E2 15565.564} C_VEL
LIN {X 0,Y 297.157,Z 691.088,A -85,B 0,C 180,E1 15569.282,E2 15569.282} C_VEL
LIN {X 0,Y 301.245,Z 663.542,A -85,B 0,C 180,E1 15572.243,E2 15572.243} C_VEL
LIN {X 0,Y 304.063,Z 634.741,A -85,B 0,C 180,E1 15573.999,E2 15573.999} C_VEL
LIN {X 0,Y 305.025,Z 587.313,A -85,B 0,C 180,E1 15575.345,E2 15575.345} C_VEL
LIN {X 0,Y 292.85,Z 552.659,A -85,B 0,C 180,E1 15577.633,E2 15577.633} C_VEL
LIN {X 0,Y 283.041,Z 529.66,A -85,B 0,C 180,E1 15579.614,E2 15579.614} C_VEL
LIN {X 0,Y 282.41,Z 529.66,A -85,B 0,C 180,E1 15588.698,E2 15588.698} C_VEL
LIN {X 0,Y 282.008,Z 529.66,A -85,B 0,C 180,E1 15595.344,E2 15595.344} C_VEL
LIN {X 0,Y 281.736,Z 529.66,A -85,B 0,C 180,E1 15602.383,E2 15602.383} C_VEL
LIN {X 0,Y 281.482,Z 529.66,A -85,B 0,C 180,E1 15611.359,E2 15611.359} C_VEL
LIN {X 0,Y 281.783,Z 530.218,A -85,B 0,C 180,E1 15614.83,E2 15614.83} C_VEL
LIN {X 0,Y 302.372,Z 579.712,A -85,B 0,C 180,E1 15619.767,E2 15619.767} C_VEL
LIN {X 0,Y 311.949,Z 609.714,A -85,B 0,C 180,E1 15622.977,E2 15622.977} C_VEL
LIN {X 0,Y 305.863,Z 644.064,A -85,B 0,C 180,E1 15626.071,E2 15626.071} C_VEL
LIN {X 0,Y 299.322,Z 674.938,A -85,B 0,C 180,E1 15630.139,E2 15630.139} C_VEL
LIN {X 0,Y 293.163,Z 702.471,A -85,B 0,C 180,E1 15635.352,E2 15635.352} C_VEL
LIN {X 0,Y 288.491,Z 723.956,A -85,B 0,C 180,E1 15641.209,E2 15641.209} C_VEL
LIN {X 0,Y 285.783,Z 739.052,A -85,B 0,C 180,E1 15647.226,E2 15647.226} C_VEL
LIN {X 0,Y 284.521,Z 749.448,A -85,B 0,C 180,E1 15653.907,E2 15653.907} C_VEL
LIN {X 0,Y 284.403,Z 753.893,A -85,B 0,C 180,E1 15659.996,E2 15659.996} C_VEL
LIN {X 0,Y 284.884,Z 753.812,A -85,B 0,C 180,E1 15666.077,E2 15666.077} C_VEL
LIN {X 0,Y 286.98,Z 748.241,A -85,B 0,C 180,E1 15673.097,E2 15673.097} C_VEL
LIN {X 0,Y 291.278,Z 737.507,A -85,B 0,C 180,E1 15679.674,E2 15679.674} C_VEL
LIN {X 0,Y 298.848,Z 720.328,A -85,B 0,C 180,E1 15686.215,E2 15686.215} C_VEL
LIN {X 0,Y 310.164,Z 696.143,A -85,B 0,C 180,E1 15692.35,E2 15692.35} C_VEL
LIN {X 0,Y 325.246,Z 665.117,A -85,B 0,C 180,E1 15697.718,E2 15697.718} C_VEL
LIN {X 0,Y 342.775,Z 630.325,A -85,B 0,C 180,E1 15701.77,E2 15701.77} C_VEL
LIN {X 0,Y 345.967,Z 624.032,A -85,B 0,C 180,E1 15702.362,E2 15702.362} C_VEL
LIN {X 0,Y 346.246,Z 623.612,A -85,B 0,C 180,E1 15702.753,E2 15702.753} C_VEL
LIN {X 0,Y 344.879,Z 626.692,A -85,B 0,C 180,E1 15703.276,E2 15703.276} C_VEL
LIN {X 0,Y 327.033,Z 665.435,A -85,B 0,C 180,E1 15707.112,E2 15707.112} C_VEL
LIN {X 0,Y 310.82,Z 702.745,A -85,B 0,C 180,E1 15712.639,E2 15712.639} C_VEL
LIN {X 0,Y 298.901,Z 732.034,A -85,B 0,C 180,E1 15718.924,E2 15718.924} C_VEL
LIN {X 0,Y 290.744,Z 754.543,A -85,B 0,C 180,E1 15725.877,E2 15725.877} C_VEL
LIN {X 0,Y 286.116,Z 770.297,A -85,B 0,C 180,E1 15733.139,E2 15733.139} C_VEL
LIN {X 0,Y 284.577,Z 779.146,A -85,B 0,C 180,E1 15739.643,E2 15739.643} C_VEL
LIN {X 0,Y 284.257,Z 782.444,A -85,B 0,C 180,E1 15743.907,E2 15743.907} C_VEL
LIN {X 0,Y 284.382,Z 783.677,A -85,B 0,C 180,E1 15750.001,E2 15750.001} C_VEL
LIN {X 0,Y 284.293,Z 780.546,A -85,B 0,C 180,E1 15756.095,E2 15756.095} C_VEL
LIN {X 0,Y 284.956,Z 771.631,A -85,B 0,C 180,E1 15763.008,E2 15763.008} C_VEL
LIN {X 0,Y 287.198,Z 756.637,A -85,B 0,C 180,E1 15769.833,E2 15769.833} C_VEL
LIN {X 0,Y 291.538,Z 736.317,A -85,B 0,C 180,E1 15776.103,E2 15776.103} C_VEL
LIN {X 0,Y 297.758,Z 710.409,A -85,B 0,C 180,E1 15781.723,E2 15781.723} C_VEL
LIN {X 0,Y 304.952,Z 679.973,A -85,B 0,C 180,E1 15786.428,E2 15786.428} C_VEL
LIN {X 0,Y 312.07,Z 646.246,A -85,B 0,C 180,E1 15790.071,E2 15790.071} C_VEL
LIN {X 0,Y 316.7,Z 616.092,A -85,B 0,C 180,E1 15792.41,E2 15792.41} C_VEL
LIN {X 0,Y 315.274,Z 611.7,A -85,B 0,C 180,E1 15792.885,E2 15792.885} C_VEL
LIN {X 0,Y 309.665,Z 602.064,A -85,B 0,C 180,E1 15794.153,E2 15794.153} C_VEL
LIN {X 0,Y 298.522,Z 586.867,A -85,B 0,C 180,E1 15796.319,E2 15796.319} C_VEL
LIN {X 0,Y 275.101,Z 534.08,A -85,B 0,C 180,E1 15801.871,E2 15801.871} C_VEL
LIN {X 0,Y 273.676,Z 529.66,A -85,B 0,C 180,E1 15802.471,E2 15802.471} C_VEL
LIN {X 0,Y 273.907,Z 529.66,A -85,B 0,C 180,E1 15811.822,E2 15811.822} C_VEL
LIN {X 0,Y 274.289,Z 529.66,A -85,B 0,C 180,E1 15819.272,E2 15819.272} C_VEL
LIN {X 0,Y 274.861,Z 529.66,A -85,B 0,C 180,E1 15827.319,E2 15827.319} C_VEL
LIN {X 0,Y 275.383,Z 529.66,A -85,B 0,C 180,E1 15833.712,E2 15833.712} C_VEL
LIN {X 0,Y 275.969,Z 529.66,A -85,B 0,C 180,E1 15840.004,E2 15840.004} C_VEL
LIN {X 0,Y 275.411,Z 529.66,A -85,B 0,C 180,E1 15846.295,E2 15846.295} C_VEL
LIN {X 0,Y 274.957,Z 529.66,A -85,B 0,C 180,E1 15852.685,E2 15852.685} C_VEL
LIN {X 0,Y 274.299,Z 529.66,A -85,B 0,C 180,E1 15860.733,E2 15860.733} C_VEL
LIN {X 0,Y 274.127,Z 530.241,A -85,B 0,C 180,E1 15866.341,E2 15866.341} C_VEL
LIN {X 0,Y 292.39,Z 567.653,A -85,B 0,C 180,E1 15870.751,E2 15870.751} C_VEL
LIN {X 0,Y 302.231,Z 595.597,A -85,B 0,C 180,E1 15872.997,E2 15872.997} C_VEL
LIN {X 0,Y 300.043,Z 640.883,A -85,B 0,C 180,E1 15874.345,E2 15874.345} C_VEL
LIN {X 0,Y 296.465,Z 670.206,A -85,B 0,C 180,E1 15876.367,E2 15876.367} C_VEL
LIN {X 0,Y 291.756,Z 695.71,A -85,B 0,C 180,E1 15879.382,E2 15879.382} C_VEL
LIN {X 0,Y 286.538,Z 717.466,A -85,B 0,C 180,E1 15883.33,E2 15883.33} C_VEL
LIN {X 0,Y 281.962,Z 734.796,A -85,B 0,C 180,E1 15888.131,E2 15888.131} C_VEL
LIN {X 0,Y 278.821,Z 746.905,A -85,B 0,C 180,E1 15893.463,E2 15893.463} C_VEL
LIN {X 0,Y 276.998,Z 753.722,A -85,B 0,C 180,E1 15898.832,E2 15898.832} C_VEL
LIN {X 0,Y 275.927,Z 755.947,A -85,B 0,C 180,E1 15904.054,E2 15904.054} C_VEL
LIN {X 0,Y 276.471,Z 753.792,A -85,B 0,C 180,E1 15909.584,E2 15909.584} C_VEL
LIN {X 0,Y 278.28,Z 745.729,A -85,B 0,C 180,E1 15915.725,E2 15915.725} C_VEL
LIN {X 0,Y 281.183,Z 732.003,A -85,B 0,C 180,E1 15921.33,E2 15921.33} C_VEL
LIN {X 0,Y 285.415,Z 713.036,A -85,B 0,C 180,E1 15926.209,E2 15926.209} C_VEL
LIN {X 0,Y 290.243,Z 689.089,A -85,B 0,C 180,E1 15930.185,E2 15930.185} C_VEL
LIN {X 0,Y 294.203,Z 663.299,A -85,B 0,C 180,E1 15932.939,E2 15932.939} C_VEL
LIN {X 0,Y 297.083,Z 634.381,A -85,B 0,C 180,E1 15934.707,E2 15934.707} C_VEL
LIN {X 0,Y 298.232,Z 589.523,A -85,B 0,C 180,E1 15935.989,E2 15935.989} C_VEL
LIN {X 0,Y 286.184,Z 555.315,A -85,B 0,C 180,E1 15938.333,E2 15938.333} C_VEL
LIN {X 0,Y 275.017,Z 529.66,A -85,B 0,C 180,E1 15940.571,E2 15940.571} C_VEL
LIN {X 0,Y 274.402,Z 529.66,A -85,B 0,C 180,E1 15949.264,E2 15949.264} C_VEL
LIN {X 0,Y 273.965,Z 529.66,A -85,B 0,C 180,E1 15956.143,E2 15956.143} C_VEL
LIN {X 0,Y 273.626,Z 529.66,A -85,B 0,C 180,E1 15964.179,E2 15964.179} C_VEL
LIN {X 0,Y 273.709,Z 529.909,A -85,B 0,C 180,E1 15973.715,E2 15973.715} C_VEL
LIN {X 0,Y 294.749,Z 580.39,A -85,B 0,C 180,E1 15978.974,E2 15978.974} C_VEL
LIN {X 0,Y 304.755,Z 610.943,A -85,B 0,C 180,E1 15982.393,E2 15982.393} C_VEL
LIN {X 0,Y 298.476,Z 644.977,A -85,B 0,C 180,E1 15985.552,E2 15985.552} C_VEL
LIN {X 0,Y 291.502,Z 676.786,A -85,B 0,C 180,E1 15989.898,E2 15989.898} C_VEL
LIN {X 0,Y 285.496,Z 702.816,A -85,B 0,C 180,E1 15994.982,E2 15994.982} C_VEL
LIN {X 0,Y 280.837,Z 723.595,A -85,B 0,C 180,E1 16000.746,E2 16000.746} C_VEL
LIN {X 0,Y 277.81,Z 739.998,A -85,B 0,C 180,E1 16007.447,E2 16007.447} C_VEL
LIN {X 0,Y 276.638,Z 749.553,A -85,B 0,C 180,E1 16013.733,E2 16013.733} C_VEL
LIN {X 0,Y 276.509,Z 754.25,A -85,B 0,C 180,E1 16019.996,E2 16019.996} C_VEL
LIN {X 0,Y 277.051,Z 754.457,A -85,B 0,C 180,E1 16026.25,E2 16026.25} C_VEL
LIN {X 0,Y 279.349,Z 749.166,A -85,B 0,C 180,E1 16033.517,E2 16033.517} C_VEL
LIN {X 0,Y 284.678,Z 737.385,A -85,B 0,C 180,E1 16040.96,E2 16040.96} C_VEL
LIN {X 0,Y 293.762,Z 719.083,A -85,B 0,C 180,E1 16047.947,E2 16047.947} C_VEL
LIN {X 0,Y 306.488,Z 694.913,A -85,B 0,C 180,E1 16054.054,E2 16054.054} C_VEL
LIN {X 0,Y 323.778,Z 663.517,A -85,B 0,C 180,E1 16059.459,E2 16059.459} C_VEL
LIN {X 0,Y 338.343,Z 638.311,A -85,B 0,C 180,E1 16062.479,E2 16062.479} C_VEL
LIN {X 0,Y 337.413,Z 640.242,A -85,B 0,C 180,E1 16063.011,E2 16063.011} C_VEL
LIN {X 0,Y 319.099,Z 675.533,A -85,B 0,C 180,E1 16067.037,E2 16067.037} C_VEL
LIN {X 0,Y 302.404,Z 710.065,A -85,B 0,C 180,E1 16072.77,E2 16072.77} C_VEL
LIN {X 0,Y 289.889,Z 738.245,A -85,B 0,C 180,E1 16079.588,E2 16079.588} C_VEL
LIN {X 0,Y 282.357,Z 757.699,A -85,B 0,C 180,E1 16086.372,E2 16086.372} C_VEL
LIN {X 0,Y 277.838,Z 772.747,A -85,B 0,C 180,E1 16094.244,E2 16094.244} C_VEL
LIN {X 0,Y 276.513,Z 780.024,A -85,B 0,C 180,E1 16100.579,E2 16100.579} C_VEL
LIN {X 0,Y 276.278,Z 783.102,A -85,B 0,C 180,E1 16106.87,E2 16106.87} C_VEL
LIN {X 0,Y 276.42,Z 782.201,A -85,B 0,C 180,E1 16113.131,E2 16113.131} C_VEL
LIN {X 0,Y 276.629,Z 776.476,A -85,B 0,C 180,E1 16119.42,E2 16119.42} C_VEL
LIN {X 0,Y 278.003,Z 764.513,A -85,B 0,C 180,E1 16126.558,E2 16126.558} C_VEL
LIN {X 0,Y 281.51,Z 746.47,A -85,B 0,C 180,E1 16133.43,E2 16133.43} C_VEL
LIN {X 0,Y 287.166,Z 722.846,A -85,B 0,C 180,E1 16139.616,E2 16139.616} C_VEL
LIN {X 0,Y 294.227,Z 693.981,A -85,B 0,C 180,E1 16144.955,E2 16144.955} C_VEL
LIN {X 0,Y 301.761,Z 661.402,A -85,B 0,C 180,E1 16149.197,E2 16149.197} C_VEL
LIN {X 0,Y 308.91,Z 624.55,A -85,B 0,C 180,E1 16152.46,E2 16152.46} C_VEL
LIN {X 0,Y 309.405,Z 617.79,A -85,B 0,C 180,E1 16152.989,E2 16152.989} C_VEL
LIN {X 0,Y 298.522,Z 586.867,A -85,B 0,C 180,E1 16156.319,E2 16156.319} C_VEL
LIN {X 0,Y 289.613,Z 574.651,A -85,B 0,C 180,E1 16158.042,E2 16158.042} C_VEL
LIN {X 0,Y 280.323,Z 562.513,A -85,B 0,C 180,E1 16159.797,E2 16159.797} C_VEL
LIN {X 0,Y 265.705,Z 529.66,A -85,B 0,C 180,E1 16163.581,E2 16163.581} C_VEL
LIN {X 0,Y 266.014,Z 529.66,A -85,B 0,C 180,E1 16173.017,E2 16173.017} C_VEL
LIN {X 0,Y 266.434,Z 529.66,A -85,B 0,C 180,E1 16180.139,E2 16180.139} C_VEL
LIN {X 0,Y 266.884,Z 529.66,A -85,B 0,C 180,E1 16186.933,E2 16186.933} C_VEL
LIN {X 0,Y 267.445,Z 529.66,A -85,B 0,C 180,E1 16193.525,E2 16193.525} C_VEL
LIN {X 0,Y 268.062,Z 529.66,A -85,B 0,C 180,E1 16200.004,E2 16200.004} C_VEL
LIN {X 0,Y 267.472,Z 529.66,A -85,B 0,C 180,E1 16206.483,E2 16206.483} C_VEL
LIN {X 0,Y 266.98,Z 529.66,A -85,B 0,C 180,E1 16213.071,E2 16213.071} C_VEL
LIN {X 0,Y 266.465,Z 529.66,A -85,B 0,C 180,E1 16219.868,E2 16219.868} C_VEL
LIN {X 0,Y 266.154,Z 529.66,A -85,B 0,C 180,E1 16224.646,E2 16224.646} C_VEL
LIN {X 0,Y 268.702,Z 535.47,A -85,B 0,C 180,E1 16225.447,E2 16225.447} C_VEL
LIN {X 0,Y 284.083,Z 565.442,A -85,B 0,C 180,E1 16229.368,E2 16229.368} C_VEL
LIN {X 0,Y 295.63,Z 596.655,A -85,B 0,C 180,E1 16232.13,E2 16232.13} C_VEL
LIN {X 0,Y 293.542,Z 640.657,A -85,B 0,C 180,E1 16233.471,E2 16233.471} C_VEL
LIN {X 0,Y 290.035,Z 669.019,A -85,B 0,C 180,E1 16235.425,E2 16235.425} C_VEL
LIN {X 0,Y 285.368,Z 693.709,A -85,B 0,C 180,E1 16238.282,E2 16238.282} C_VEL
LIN {X 0,Y 279.735,Z 716.23,A -85,B 0,C 180,E1 16242.301,E2 16242.301} C_VEL
LIN {X 0,Y 274.664,Z 734.473,A -85,B 0,C 180,E1 16247.338,E2 16247.338} C_VEL
LIN {X 0,Y 271.471,Z 745.953,A -85,B 0,C 180,E1 16252.304,E2 16252.304} C_VEL
LIN {X 0,Y 269.221,Z 753.937,A -85,B 0,C 180,E1 16258.376,E2 16258.376} C_VEL
LIN {X 0,Y 268.047,Z 756.357,A -85,B 0,C 180,E1 16264.263,E2 16264.263} C_VEL
LIN {X 0,Y 268.736,Z 753.652,A -85,B 0,C 180,E1 16270.31,E2 16270.31} C_VEL
LIN {X 0,Y 270.665,Z 744.923,A -85,B 0,C 180,E1 16276.599,E2 16276.599} C_VEL
LIN {X 0,Y 273.881,Z 731.14,A -85,B 0,C 180,E1 16282.138,E2 16282.138} C_VEL
LIN {X 0,Y 278.136,Z 712.648,A -85,B 0,C 180,E1 16286.889,E2 16286.889} C_VEL
LIN {X 0,Y 282.934,Z 689.748,A -85,B 0,C 180,E1 16290.763,E2 16290.763} C_VEL
LIN {X 0,Y 287.227,Z 662.938,A -85,B 0,C 180,E1 16293.676,E2 16293.676} C_VEL
LIN {X 0,Y 290.162,Z 633.66,A -85,B 0,C 180,E1 16295.466,E2 16295.466} C_VEL
LIN {X 0,Y 291.059,Z 590.341,A -85,B 0,C 180,E1 16296.747,E2 16296.747} C_VEL
LIN {X 0,Y 279.473,Z 557.873,A -85,B 0,C 180,E1 16299.081,E2 16299.081} C_VEL
LIN {X 0,Y 267.013,Z 529.66,A -85,B 0,C 180,E1 16301.788,E2 16301.788} C_VEL
LIN {X 0,Y 266.432,Z 529.66,A -85,B 0,C 180,E1 16309.865,E2 16309.865} C_VEL
LIN {X 0,Y 265.987,Z 529.66,A -85,B 0,C 180,E1 16316.99,E2 16316.99} C_VEL
LIN {X 0,Y 265.677,Z 529.66,A -85,B 0,C 180,E1 16324.608,E2 16324.608} C_VEL
LIN {X 0,Y 265.687,Z 529.66,A -85,B 0,C 180,E1 16332.543,E2 16332.543} C_VEL
LIN {X 0,Y 286.984,Z 580.566,A -85,B 0,C 180,E1 16338.101,E2 16338.101} C_VEL
LIN {X 0,Y 297.375,Z 613.301,A -85,B 0,C 180,E1 16341.881,E2 16341.881} C_VEL
LIN {X 0,Y 290.574,Z 648.439,A -85,B 0,C 180,E1 16345.322,E2 16345.322} C_VEL
LIN {X 0,Y 283.431,Z 679.662,A -85,B 0,C 180,E1 16349.833,E2 16349.833} C_VEL
LIN {X 0,Y 277.355,Z 704.986,A -85,B 0,C 180,E1 16355.057,E2 16355.057} C_VEL
LIN {X 0,Y 272.723,Z 725.464,A -85,B 0,C 180,E1 16361.026,E2 16361.026} C_VEL
LIN {X 0,Y 270.012,Z 739.794,A -85,B 0,C 180,E1 16367.078,E2 16367.078} C_VEL
LIN {X 0,Y 268.77,Z 749.631,A -85,B 0,C 180,E1 16373.548,E2 16373.548} C_VEL
LIN {X 0,Y 268.618,Z 754.593,A -85,B 0,C 180,E1 16379.996,E2 16379.996} C_VEL
LIN {X 0,Y 269.197,Z 755.074,A -85,B 0,C 180,E1 16386.433,E2 16386.433} C_VEL
LIN {X 0,Y 271.707,Z 750.197,A -85,B 0,C 180,E1 16393.904,E2 16393.904} C_VEL
LIN {X 0,Y 277.444,Z 738.99,A -85,B 0,C 180,E1 16401.534,E2 16401.534} C_VEL
LIN {X 0,Y 287.131,Z 721.516,A -85,B 0,C 180,E1 16408.636,E2 16408.636} C_VEL
LIN {X 0,Y 301.471,Z 697.161,A -85,B 0,C 180,E1 16415.138,E2 16415.138} C_VEL
LIN {X 0,Y 321.002,Z 665.961,A -85,B 0,C 180,E1 16420.706,E2 16420.706} C_VEL
LIN {X 0,Y 329.541,Z 652.934,A -85,B 0,C 180,E1 16422.422,E2 16422.422} C_VEL
LIN {X 0,Y 328.599,Z 654.624,A -85,B 0,C 180,E1 16422.957,E2 16422.957} C_VEL
LIN {X 0,Y 309.41,Z 687.953,A -85,B 0,C 180,E1 16427.417,E2 16427.417} C_VEL
LIN {X 0,Y 292.35,Z 720.252,A -85,B 0,C 180,E1 16433.684,E2 16433.684} C_VEL
LIN {X 0,Y 280.482,Z 744.955,A -85,B 0,C 180,E1 16440.642,E2 16440.642} C_VEL
LIN {X 0,Y 273.043,Z 763.184,A -85,B 0,C 180,E1 16448.098,E2 16448.098} C_VEL
LIN {X 0,Y 269.572,Z 774.847,A -85,B 0,C 180,E1 16455.412,E2 16455.412} C_VEL
LIN {X 0,Y 268.645,Z 779.721,A -85,B 0,C 180,E1 16460.3,E2 16460.3} C_VEL
LIN {X 0,Y 268.379,Z 782.658,A -85,B 0,C 180,E1 16466.778,E2 16466.778} C_VEL
LIN {X 0,Y 268.516,Z 781.827,A -85,B 0,C 180,E1 16473.223,E2 16473.223} C_VEL
LIN {X 0,Y 268.662,Z 777.07,A -85,B 0,C 180,E1 16478.887,E2 16478.887} C_VEL
LIN {X 0,Y 270.192,Z 763.721,A -85,B 0,C 180,E1 16486.862,E2 16486.862} C_VEL
LIN {X 0,Y 273.738,Z 746.145,A -85,B 0,C 180,E1 16493.701,E2 16493.701} C_VEL
LIN {X 0,Y 279.291,Z 723.569,A -85,B 0,C 180,E1 16499.807,E2 16499.807} C_VEL
LIN {X 0,Y 286.647,Z 694.463,A -85,B 0,C 180,E1 16505.387,E2 16505.387} C_VEL
LIN {X 0,Y 294.486,Z 661.646,A -85,B 0,C 180,E1 16509.777,E2 16509.777} C_VEL
LIN {X 0,Y 301.75,Z 625.47,A -85,B 0,C 180,E1 16513.076,E2 16513.076} C_VEL
LIN {X 0,Y 302.103,Z 619.648,A -85,B 0,C 180,E1 16513.566,E2 16513.566} C_VEL
LIN {X 0,Y 289.05,Z 583.036,A -85,B 0,C 180,E1 16517.634,E2 16517.634} C_VEL
LIN {X 0,Y 280.323,Z 562.513,A -85,B 0,C 180,E1 16519.797,E2 16519.797} C_VEL
LIN {X 0,Y 271.183,Z 550.437,A -85,B 0,C 180,E1 16521.618,E2 16521.618} C_VEL
LIN {X 0,Y 261.52,Z 538.966,A -85,B 0,C 180,E1 16523.625,E2 16523.625} C_VEL
LIN {X 0,Y 257.785,Z 529.66,A -85,B 0,C 180,E1 16524.827,E2 16524.827} C_VEL
LIN {X 0,Y 257.957,Z 529.66,A -85,B 0,C 180,E1 16532.102,E2 16532.102} C_VEL
LIN {X 0,Y 258.415,Z 529.66,A -85,B 0,C 180,E1 16539.495,E2 16539.495} C_VEL
LIN {X 0,Y 258.943,Z 529.66,A -85,B 0,C 180,E1 16546.525,E2 16546.525} C_VEL
LIN {X 0,Y 259.495,Z 529.66,A -85,B 0,C 180,E1 16553.326,E2 16553.326} C_VEL
LIN {X 0,Y 260.155,Z 529.66,A -85,B 0,C 180,E1 16560.004,E2 16560.004} C_VEL
LIN {X 0,Y 259.357,Z 529.66,A -85,B 0,C 180,E1 16568.459,E2 16568.459} C_VEL
LIN {X 0,Y 258.747,Z 529.66,A -85,B 0,C 180,E1 16576.958,E2 16576.958} C_VEL
LIN {X 0,Y 258.384,Z 530.472,A -85,B 0,C 180,E1 16582.949,E2 16582.949} C_VEL
LIN {X 0,Y 276.086,Z 563.97,A -85,B 0,C 180,E1 16587.934,E2 16587.934} C_VEL
LIN {X 0,Y 288.258,Z 595.527,A -85,B 0,C 180,E1 16591.018,E2 16591.018} C_VEL
LIN {X 0,Y 289.122,Z 602.991,A -85,B 0,C 180,E1 16591.388,E2 16591.388} C_VEL
LIN {X 0,Y 286.874,Z 642.963,A -85,B 0,C 180,E1 16592.686,E2 16592.686} C_VEL
LIN {X 0,Y 282.957,Z 671.685,A -85,B 0,C 180,E1 16594.779,E2 16594.779} C_VEL
LIN {X 0,Y 277.652,Z 697.678,A -85,B 0,C 180,E1 16598.031,E2 16598.031} C_VEL
LIN {X 0,Y 271.974,Z 718.869,A -85,B 0,C 180,E1 16602.109,E2 16602.109} C_VEL
LIN {X 0,Y 266.722,Z 736.498,A -85,B 0,C 180,E1 16607.353,E2 16607.353} C_VEL
LIN {X 0,Y 263.073,Z 748.927,A -85,B 0,C 180,E1 16613.428,E2 16613.428} C_VEL
LIN {X 0,Y 261.229,Z 754.75,A -85,B 0,C 180,E1 16618.674,E2 16618.674} C_VEL
LIN {X 0,Y 260.308,Z 756.533,A -85,B 0,C 180,E1 16622.369,E2 16622.369} C_VEL
LIN {X 0,Y 260.358,Z 755.663,A -85,B 0,C 180,E1 16628.033,E2 16628.033} C_VEL
LIN {X 0,Y 261.906,Z 749.81,A -85,B 0,C 180,E1 16634.115,E2 16634.115} C_VEL
LIN {X 0,Y 264.664,Z 738.213,A -85,B 0,C 180,E1 16640.15,E2 16640.15} C_VEL
LIN {X 0,Y 268.841,Z 721.021,A -85,B 0,C 180,E1 16645.572,E2 16645.572} C_VEL
LIN {X 0,Y 273.808,Z 699.418,A -85,B 0,C 180,E1 16649.999,E2 16649.999} C_VEL
LIN {X 0,Y 278.563,Z 674.612,A -85,B 0,C 180,E1 16653.291,E2 16653.291} C_VEL
LIN {X 0,Y 282.253,Z 645.729,A -85,B 0,C 180,E1 16655.623,E2 16655.623} C_VEL
LIN {X 0,Y 284.165,Z 614.157,A -85,B 0,C 180,E1 16656.826,E2 16656.826} C_VEL
LIN {X 0,Y 284.231,Z 592.307,A -85,B 0,C 180,E1 16657.465,E2 16657.465} C_VEL
LIN {X 0,Y 272.921,Z 560.598,A -85,B 0,C 180,E1 16659.844,E2 16659.844} C_VEL
LIN {X 0,Y 259.024,Z 529.66,A -85,B 0,C 180,E1 16662.923,E2 16662.923} C_VEL
LIN {X 0,Y 258.384,Z 529.66,A -85,B 0,C 180,E1 16670.855,E2 16670.855} C_VEL
LIN {X 0,Y 257.868,Z 529.66,A -85,B 0,C 180,E1 16678.618,E2 16678.618} C_VEL
LIN {X 0,Y 257.71,Z 529.66,A -85,B 0,C 180,E1 16685.839,E2 16685.839} C_VEL
LIN {X 0,Y 257.647,Z 529.66,A -85,B 0,C 180,E1 16691.314,E2 16691.314} C_VEL
LIN {X 0,Y 279.055,Z 580.603,A -85,B 0,C 180,E1 16697.17,E2 16697.17} C_VEL
LIN {X 0,Y 290.11,Z 614.651,A -85,B 0,C 180,E1 16701.278,E2 16701.278} C_VEL
LIN {X 0,Y 283.259,Z 648.874,A -85,B 0,C 180,E1 16704.73,E2 16704.73} C_VEL
LIN {X 0,Y 275.893,Z 680.212,A -85,B 0,C 180,E1 16709.375,E2 16709.375} C_VEL
LIN {X 0,Y 269.62,Z 705.511,A -85,B 0,C 180,E1 16714.734,E2 16714.734} C_VEL
LIN {X 0,Y 264.635,Z 727.097,A -85,B 0,C 180,E1 16721.288,E2 16721.288} C_VEL
LIN {X 0,Y 261.743,Z 742.901,A -85,B 0,C 180,E1 16728.537,E2 16728.537} C_VEL
LIN {X 0,Y 260.748,Z 751.46,A -85,B 0,C 180,E1 16735.016,E2 16735.016} C_VEL
LIN {X 0,Y 260.722,Z 754.925,A -85,B 0,C 180,E1 16739.996,E2 16739.996} C_VEL
LIN {X 0,Y 261.371,Z 755.699,A -85,B 0,C 180,E1 16746.626,E2 16746.626} C_VEL
LIN {X 0,Y 263.523,Z 752.213,A -85,B 0,C 180,E1 16753.236,E2 16753.236} C_VEL
LIN {X 0,Y 268.662,Z 743.325,A -85,B 0,C 180,E1 16760.546,E2 16760.546} C_VEL
LIN {X 0,Y 278.648,Z 727.024,A -85,B 0,C 180,E1 16768.279,E2 16768.279} C_VEL
LIN {X 0,Y 293.903,Z 703.748,A -85,B 0,C 180,E1 16775.277,E2 16775.277} C_VEL
LIN {X 0,Y 313.749,Z 675.434,A -85,B 0,C 180,E1 16780.937,E2 16780.937} C_VEL
LIN {X 0,Y 321.01,Z 665.539,A -85,B 0,C 180,E1 16782.427,E2 16782.427} C_VEL
LIN {X 0,Y 318.009,Z 670.158,A -85,B 0,C 180,E1 16783.251,E2 16783.251} C_VEL
LIN {X 0,Y 296.971,Z 703.506,A -85,B 0,C 180,E1 16788.659,E2 16788.659} C_VEL
LIN {X 0,Y 280.466,Z 732.643,A -85,B 0,C 180,E1 16795.604,E2 16795.604} C_VEL
LIN {X 0,Y 269.379,Z 754.832,A -85,B 0,C 180,E1 16803.377,E2 16803.377} C_VEL
LIN {X 0,Y 263.539,Z 768.969,A -85,B 0,C 180,E1 16810.723,E2 16810.723} C_VEL
LIN {X 0,Y 261.022,Z 778.065,A -85,B 0,C 180,E1 16818.292,E2 16818.292} C_VEL
LIN {X 0,Y 260.58,Z 781.3,A -85,B 0,C 180,E1 16823.351,E2 16823.351} C_VEL
LIN {X 0,Y 260.723,Z 782.019,A -85,B 0,C 180,E1 16830.001,E2 16830.001} C_VEL
LIN {X 0,Y 260.576,Z 780.615,A -85,B 0,C 180,E1 16834.985,E2 16834.985} C_VEL
LIN {X 0,Y 261.073,Z 774.668,A -85,B 0,C 180,E1 16840.734,E2 16840.734} C_VEL
LIN {X 0,Y 263.322,Z 757.567,A -85,B 0,C 180,E1 16849.595,E2 16849.595} C_VEL
LIN {X 0,Y 267.617,Z 738.35,A -85,B 0,C 180,E1 16856.29,E2 16856.29} C_VEL
LIN {X 0,Y 274.36,Z 712.886,A -85,B 0,C 180,E1 16862.523,E2 16862.523} C_VEL
LIN {X 0,Y 282.21,Z 682.639,A -85,B 0,C 180,E1 16867.705,E2 16867.705} C_VEL
LIN {X 0,Y 290.168,Z 648.735,A -85,B 0,C 180,E1 16871.762,E2 16871.762} C_VEL
LIN {X 0,Y 295.063,Z 622.446,A -85,B 0,C 180,E1 16874.02,E2 16874.02} C_VEL
LIN {X 0,Y 282.275,Z 585.889,A -85,B 0,C 180,E1 16878.282,E2 16878.282} C_VEL
LIN {X 0,Y 261.52,Z 538.966,A -85,B 0,C 180,E1 16883.625,E2 16883.625} C_VEL
LIN {X 0,Y 254.419,Z 532.125,A -85,B 0,C 180,E1 16885.319,E2 16885.319} C_VEL
LIN {X 0,Y 250.001,Z 529.707,A -85,B 0,C 180,E1 16887.41,E2 16887.41} C_VEL
LIN {X 0,Y 249.87,Z 529.66,A -85,B 0,C 180,E1 16887.752,E2 16887.752} C_VEL
LIN {X 0,Y 250.177,Z 529.66,A -85,B 0,C 180,E1 16895.031,E2 16895.031} C_VEL
LIN {X 0,Y 250.68,Z 529.66,A -85,B 0,C 180,E1 16902.489,E2 16902.489} C_VEL
LIN {X 0,Y 251.244,Z 529.66,A -85,B 0,C 180,E1 16909.624,E2 16909.624} C_VEL
LIN {X 0,Y 251.972,Z 529.66,A -85,B 0,C 180,E1 16916.571,E2 16916.571} C_VEL
LIN {X 0,Y 251.942,Z 529.66,A -85,B 0,C 180,E1 16923.438,E2 16923.438} C_VEL
LIN {X 0,Y 251.321,Z 529.66,A -85,B 0,C 180,E1 16930.382,E2 16930.382} C_VEL
LIN {X 0,Y 250.558,Z 529.66,A -85,B 0,C 180,E1 16939.349,E2 16939.349} C_VEL
LIN {X 0,Y 250.549,Z 530.331,A -85,B 0,C 180,E1 16940.958,E2 16940.958} C_VEL
LIN {X 0,Y 253.44,Z 535.864,A -85,B 0,C 180,E1 16941.966,E2 16941.966} C_VEL
LIN {X 0,Y 268.906,Z 564.281,A -85,B 0,C 180,E1 16946.592,E2 16946.592} C_VEL
LIN {X 0,Y 281.328,Z 595.52,A -85,B 0,C 180,E1 16949.93,E2 16949.93} C_VEL
LIN {X 0,Y 282.919,Z 600.649,A -85,B 0,C 180,E1 16950.357,E2 16950.357} C_VEL
LIN {X 0,Y 280.527,Z 642.875,A -85,B 0,C 180,E1 16951.729,E2 16951.729} C_VEL
LIN {X 0,Y 276.527,Z 671.453,A -85,B 0,C 180,E1 16953.827,E2 16953.827} C_VEL
LIN {X 0,Y 270.964,Z 697.484,A -85,B 0,C 180,E1 16957.11,E2 16957.11} C_VEL
LIN {X 0,Y 265.085,Z 718.408,A -85,B 0,C 180,E1 16961.163,E2 16961.163} C_VEL
LIN {X 0,Y 259.619,Z 735.928,A -85,B 0,C 180,E1 16966.366,E2 16966.366} C_VEL
LIN {X 0,Y 255.757,Z 748.123,A -85,B 0,C 180,E1 16972.202,E2 16972.202} C_VEL
LIN {X 0,Y 253.664,Z 754.56,A -85,B 0,C 180,E1 16977.628,E2 16977.628} C_VEL
LIN {X 0,Y 252.239,Z 757.12,A -85,B 0,C 180,E1 16983.822,E2 16983.822} C_VEL
LIN {X 0,Y 253.029,Z 754.173,A -85,B 0,C 180,E1 16990.759,E2 16990.759} C_VEL
LIN {X 0,Y 255.019,Z 745.98,A -85,B 0,C 180,E1 16996.995,E2 16996.995} C_VEL
LIN {X 0,Y 258.537,Z 732.275,A -85,B 0,C 180,E1 17002.883,E2 17002.883} C_VEL
LIN {X 0,Y 263.189,Z 713.803,A -85,B 0,C 180,E1 17007.932,E2 17007.932} C_VEL
LIN {X 0,Y 268.395,Z 690.953,A -85,B 0,C 180,E1 17012.012,E2 17012.012} C_VEL
LIN {X 0,Y 273.078,Z 664.111,A -85,B 0,C 180,E1 17015.08,E2 17015.08} C_VEL
LIN {X 0,Y 276.262,Z 635.06,A -85,B 0,C 180,E1 17016.953,E2 17016.953} C_VEL
LIN {X 0,Y 277.406,Z 594.199,A -85,B 0,C 180,E1 17018.224,E2 17018.224} C_VEL
LIN {X 0,Y 266.164,Z 562.753,A -85,B 0,C 180,E1 17020.685,E2 17020.685} C_VEL
LIN {X 0,Y 250.932,Z 529.66,A -85,B 0,C 180,E1 17024.134,E2 17024.134} C_VEL
LIN {X 0,Y 250.435,Z 529.66,A -85,B 0,C 180,E1 17031.193,E2 17031.193} C_VEL
LIN {X 0,Y 249.954,Z 529.66,A -85,B 0,C 180,E1 17038.878,E2 17038.878} C_VEL
LIN {X 0,Y 249.621,Z 529.66,A -85,B 0,C 180,E1 17047.192,E2 17047.192} C_VEL
LIN {X 0,Y 249.753,Z 530.476,A -85,B 0,C 180,E1 17050.155,E2 17050.155} C_VEL
LIN {X 0,Y 269.818,Z 577.077,A -85,B 0,C 180,E1 17055.769,E2 17055.769} C_VEL
LIN {X 0,Y 280.941,Z 610.02,A -85,B 0,C 180,E1 17059.864,E2 17059.864} C_VEL
LIN {X 0,Y 282.487,Z 617.933,A -85,B 0,C 180,E1 17060.835,E2 17060.835} C_VEL
LIN {X 0,Y 275.248,Z 652.36,A -85,B 0,C 180,E1 17064.514,E2 17064.514} C_VEL
LIN {X 0,Y 267.812,Z 682.863,A -85,B 0,C 180,E1 17069.29,E2 17069.29} C_VEL
LIN {X 0,Y 261.148,Z 709.146,A -85,B 0,C 180,E1 17075.229,E2 17075.229} C_VEL
LIN {X 0,Y 256.305,Z 729.754,A -85,B 0,C 180,E1 17082,E2 17082} C_VEL
LIN {X 0,Y 253.745,Z 743.912,A -85,B 0,C 180,E1 17088.946,E2 17088.946} C_VEL
LIN {X 0,Y 252.87,Z 751.56,A -85,B 0,C 180,E1 17094.86,E2 17094.86} C_VEL
LIN {X 0,Y 252.826,Z 755.247,A -85,B 0,C 180,E1 17099.995,E2 17099.995} C_VEL
LIN {X 0,Y 253.528,Z 756.335,A -85,B 0,C 180,E1 17106.832,E2 17106.832} C_VEL
LIN {X 0,Y 255.859,Z 753.212,A -85,B 0,C 180,E1 17113.64,E2 17113.64} C_VEL
LIN {X 0,Y 262.241,Z 743.58,A -85,B 0,C 180,E1 17121.959,E2 17121.959} C_VEL
LIN {X 0,Y 273.454,Z 727.503,A -85,B 0,C 180,E1 17129.773,E2 17129.773} C_VEL
LIN {X 0,Y 291.059,Z 703.695,A -85,B 0,C 180,E1 17137.058,E2 17137.058} C_VEL
LIN {X 0,Y 312.723,Z 676.67,A -85,B 0,C 180,E1 17142.491,E2 17142.491} C_VEL
LIN {X 0,Y 288.532,Z 711.116,A -85,B 0,C 180,E1 17148.681,E2 17148.681} C_VEL
LIN {X 0,Y 271.252,Z 738.944,A -85,B 0,C 180,E1 17156.201,E2 17156.201} C_VEL
LIN {X 0,Y 260.655,Z 758.584,A -85,B 0,C 180,E1 17164.073,E2 17164.073} C_VEL
LIN {X 0,Y 254.64,Z 772.65,A -85,B 0,C 180,E1 17172.766,E2 17172.766} C_VEL
LIN {X 0,Y 252.921,Z 779.136,A -85,B 0,C 180,E1 17179.691,E2 17179.691} C_VEL
LIN {X 0,Y 252.584,Z 781.671,A -85,B 0,C 180,E1 17186.576,E2 17186.576} C_VEL
LIN {X 0,Y 252.71,Z 781.09,A -85,B 0,C 180,E1 17193.425,E2 17193.425} C_VEL
LIN {X 0,Y 252.962,Z 776.461,A -85,B 0,C 180,E1 17199.443,E2 17199.443} C_VEL
LIN {X 0,Y 253.992,Z 766.752,A -85,B 0,C 180,E1 17205.508,E2 17205.508} C_VEL
LIN {X 0,Y 258.456,Z 744.35,A -85,B 0,C 180,E1 17214.607,E2 17214.607} C_VEL
LIN {X 0,Y 264.67,Z 720.628,A -85,B 0,C 180,E1 17221.226,E2 17221.226} C_VEL
LIN {X 0,Y 272.328,Z 692.05,A -85,B 0,C 180,E1 17226.814,E2 17226.814} C_VEL
LIN {X 0,Y 280.753,Z 658.541,A -85,B 0,C 180,E1 17231.392,E2 17231.392} C_VEL
LIN {X 0,Y 287.784,Z 624.427,A -85,B 0,C 180,E1 17234.585,E2 17234.585} C_VEL
LIN {X 0,Y 275.543,Z 588.726,A -85,B 0,C 180,E1 17238.922,E2 17238.922} C_VEL
LIN {X 0,Y 255.85,Z 543.737,A -85,B 0,C 180,E1 17244.237,E2 17244.237} C_VEL
LIN {X 0,Y 249.829,Z 529.66,A -85,B 0,C 180,E1 17246.089,E2 17246.089} C_VEL
LIN {X 0,Y 249.87,Z 529.66,A -85,B 0,C 180,E1 17247.752,E2 17247.752} C_VEL
LIN {X 0,Y 247.279,Z 529.66,A -85,B 0,C 180,E1 17250.712,E2 17250.712} C_VEL
LIN {X 0,Y 242.131,Z 529.66,A -85,B 0,C 180,E1 17255.739,E2 17255.739} C_VEL
LIN {X 0,Y 242.667,Z 529.66,A -85,B 0,C 180,E1 17261.891,E2 17261.891} C_VEL
LIN {X 0,Y 243.268,Z 529.66,A -85,B 0,C 180,E1 17269.28,E2 17269.28} C_VEL
LIN {X 0,Y 244.033,Z 529.66,A -85,B 0,C 180,E1 17276.46,E2 17276.46} C_VEL
LIN {X 0,Y 244.009,Z 529.66,A -85,B 0,C 180,E1 17283.55,E2 17283.55} C_VEL
LIN {X 0,Y 243.372,Z 529.66,A -85,B 0,C 180,E1 17290.725,E2 17290.725} C_VEL
LIN {X 0,Y 242.714,Z 529.66,A -85,B 0,C 180,E1 17298.64,E2 17298.64} C_VEL
LIN {X 0,Y 245.087,Z 535.372,A -85,B 0,C 180,E1 17299.669,E2 17299.669} C_VEL
LIN {X 0,Y 258.728,Z 558.558,A -85,B 0,C 180,E1 17304.215,E2 17304.215} C_VEL
LIN {X 0,Y 271.09,Z 586.217,A -85,B 0,C 180,E1 17307.822,E2 17307.822} C_VEL
LIN {X 0,Y 276.681,Z 602.697,A -85,B 0,C 180,E1 17309.401,E2 17309.401} C_VEL
LIN {X 0,Y 274.213,Z 643.396,A -85,B 0,C 180,E1 17310.761,E2 17310.761} C_VEL
LIN {X 0,Y 270.053,Z 671.849,A -85,B 0,C 180,E1 17312.886,E2 17312.886} C_VEL
LIN {X 0,Y 264.144,Z 698.149,A -85,B 0,C 180,E1 17316.269,E2 17316.269} C_VEL
LIN {X 0,Y 257.897,Z 719.243,A -85,B 0,C 180,E1 17320.476,E2 17320.476} C_VEL
LIN {X 0,Y 252.042,Z 736.894,A -85,B 0,C 180,E1 17325.932,E2 17325.932} C_VEL
LIN {X 0,Y 247.72,Z 749.639,A -85,B 0,C 180,E1 17332.47,E2 17332.47} C_VEL
LIN {X 0,Y 245.591,Z 755.539,A -85,B 0,C 180,E1 17338.107,E2 17338.107} C_VEL
LIN {X 0,Y 244.344,Z 757.492,A -85,B 0,C 180,E1 17344.385,E2 17344.385} C_VEL
LIN {X 0,Y 245.005,Z 755.099,A -85,B 0,C 180,E1 17350.198,E2 17350.198} C_VEL
LIN {X 0,Y 247.064,Z 747.274,A -85,B 0,C 180,E1 17356.764,E2 17356.764} C_VEL
LIN {X 0,Y 250.729,Z 733.397,A -85,B 0,C 180,E1 17363.085,E2 17363.085} C_VEL
LIN {X 0,Y 255.661,Z 714.729,A -85,B 0,C 180,E1 17368.417,E2 17368.417} C_VEL
LIN {X 0,Y 261.165,Z 691.535,A -85,B 0,C 180,E1 17372.689,E2 17372.689} C_VEL
LIN {X 0,Y 266.088,Z 664.401,A -85,B 0,C 180,E1 17375.862,E2 17375.862} C_VEL
LIN {X 0,Y 269.44,Z 634.803,A -85,B 0,C 180,E1 17377.792,E2 17377.792} C_VEL
LIN {X 0,Y 270.526,Z 595.717,A -85,B 0,C 180,E1 17379.039,E2 17379.039} C_VEL
LIN {X 0,Y 258.843,Z 563.632,A -85,B 0,C 180,E1 17381.705,E2 17381.705} C_VEL
LIN {X 0,Y 242.886,Z 529.66,A -85,B 0,C 180,E1 17385.598,E2 17385.598} C_VEL
LIN {X 0,Y 242.39,Z 529.66,A -85,B 0,C 180,E1 17391.932,E2 17391.932} C_VEL
LIN {X 0,Y 241.951,Z 529.66,A -85,B 0,C 180,E1 17399.928,E2 17399.928} C_VEL
LIN {X 0,Y 241.712,Z 529.66,A -85,B 0,C 180,E1 17408.757,E2 17408.757} C_VEL
LIN {X 0,Y 262.415,Z 578.158,A -85,B 0,C 180,E1 17414.891,E2 17414.891} C_VEL
LIN {X 0,Y 273.274,Z 610.619,A -85,B 0,C 180,E1 17419.076,E2 17419.076} C_VEL
LIN {X 0,Y 275.133,Z 619.794,A -85,B 0,C 180,E1 17420.258,E2 17420.258} C_VEL
LIN {X 0,Y 267.476,Z 654.77,A -85,B 0,C 180,E1 17424.17,E2 17424.17} C_VEL
LIN {X 0,Y 259.728,Z 685.287,A -85,B 0,C 180,E1 17429.198,E2 17429.198} C_VEL
LIN {X 0,Y 253.006,Z 711.034,A -85,B 0,C 180,E1 17435.319,E2 17435.319} C_VEL
LIN {X 0,Y 248.198,Z 731.238,A -85,B 0,C 180,E1 17442.298,E2 17442.298} C_VEL
LIN {X 0,Y 245.751,Z 744.878,A -85,B 0,C 180,E1 17449.38,E2 17449.38} C_VEL
LIN {X 0,Y 244.822,Z 753.169,A -85,B 0,C 180,E1 17456.462,E2 17456.462} C_VEL
LIN {X 0,Y 245.129,Z 756.783,A -85,B 0,C 180,E1 17463.525,E2 17463.525} C_VEL
LIN {X 0,Y 246.713,Z 756.095,A -85,B 0,C 180,E1 17470.568,E2 17470.568} C_VEL
LIN {X 0,Y 251.771,Z 749.545,A -85,B 0,C 180,E1 17479.242,E2 17479.242} C_VEL
LIN {X 0,Y 261.585,Z 736.856,A -85,B 0,C 180,E1 17487.478,E2 17487.478} C_VEL
LIN {X 0,Y 278.214,Z 716.398,A -85,B 0,C 180,E1 17495.442,E2 17495.442} C_VEL
LIN {X 0,Y 300.193,Z 691.351,A -85,B 0,C 180,E1 17501.687,E2 17501.687} C_VEL
LIN {X 0,Y 303.161,Z 688.093,A -85,B 0,C 180,E1 17502.332,E2 17502.332} C_VEL
LIN {X 0,Y 299.194,Z 693.107,A -85,B 0,C 180,E1 17503.412,E2 17503.412} C_VEL
LIN {X 0,Y 276.904,Z 722.427,A -85,B 0,C 180,E1 17509.784,E2 17509.784} C_VEL
LIN {X 0,Y 259.458,Z 748.712,A -85,B 0,C 180,E1 17518.439,E2 17518.439} C_VEL
LIN {X 0,Y 250.119,Z 765.52,A -85,B 0,C 180,E1 17526.913,E2 17526.913} C_VEL
LIN {X 0,Y 245.76,Z 776.241,A -85,B 0,C 180,E1 17535.784,E2 17535.784} C_VEL
LIN {X 0,Y 244.763,Z 780.56,A -85,B 0,C 180,E1 17542.919,E2 17542.919} C_VEL
LIN {X 0,Y 244.93,Z 781.2,A -85,B 0,C 180,E1 17550.002,E2 17550.002} C_VEL
LIN {X 0,Y 244.805,Z 779.919,A -85,B 0,C 180,E1 17555.307,E2 17555.307} C_VEL
LIN {X 0,Y 245.334,Z 773.963,A -85,B 0,C 180,E1 17561.533,E2 17561.533} C_VEL
LIN {X 0,Y 246.819,Z 762.733,A -85,B 0,C 180,E1 17567.801,E2 17567.801} C_VEL
LIN {X 0,Y 252.526,Z 736.382,A -85,B 0,C 180,E1 17577.345,E2 17577.345} C_VEL
LIN {X 0,Y 259.594,Z 711.057,A -85,B 0,C 180,E1 17583.771,E2 17583.771} C_VEL
LIN {X 0,Y 267.824,Z 681.18,A -85,B 0,C 180,E1 17589.076,E2 17589.076} C_VEL
LIN {X 0,Y 276.35,Z 646.775,A -85,B 0,C 180,E1 17593.313,E2 17593.313} C_VEL
LIN {X 0,Y 280.28,Z 625.494,A -85,B 0,C 180,E1 17595.277,E2 17595.277} C_VEL
LIN {X 0,Y 268.051,Z 589.85,A -85,B 0,C 180,E1 17599.793,E2 17599.793} C_VEL
LIN {X 0,Y 250.065,Z 548.229,A -85,B 0,C 180,E1 17604.896,E2 17604.896} C_VEL
LIN {X 0,Y 241.956,Z 529.66,A -85,B 0,C 180,E1 17607.53,E2 17607.53} C_VEL
LIN {X 0,Y 242.131,Z 529.66,A -85,B 0,C 180,E1 17615.739,E2 17615.739} C_VEL
LIN {X 0,Y 239.743,Z 529.66,A -85,B 0,C 180,E1 17618.809,E2 17618.809} C_VEL
LIN {X 0,Y 234.799,Z 529.66,A -85,B 0,C 180,E1 17624.03,E2 17624.03} C_VEL
LIN {X 0,Y 235.673,Z 529.66,A -85,B 0,C 180,E1 17632.648,E2 17632.648} C_VEL
LIN {X 0,Y 236.441,Z 529.66,A -85,B 0,C 180,E1 17640.005,E2 17640.005} C_VEL
LIN {X 0,Y 235.749,Z 529.66,A -85,B 0,C 180,E1 17647.36,E2 17647.36} C_VEL
LIN {X 0,Y 234.922,Z 530.064,A -85,B 0,C 180,E1 17656.104,E2 17656.104} C_VEL
LIN {X 0,Y 237.208,Z 535.304,A -85,B 0,C 180,E1 17657.202,E2 17657.202} C_VEL
LIN {X 0,Y 243.003,Z 544.152,A -85,B 0,C 180,E1 17659.493,E2 17659.493} C_VEL
LIN {X 0,Y 256.994,Z 569.488,A -85,B 0,C 180,E1 17664.273,E2 17664.273} C_VEL
LIN {X 0,Y 268.132,Z 597.084,A -85,B 0,C 180,E1 17667.669,E2 17667.669} C_VEL
LIN {X 0,Y 270.546,Z 605.403,A -85,B 0,C 180,E1 17668.418,E2 17668.418} C_VEL
LIN {X 0,Y 268.058,Z 643.591,A -85,B 0,C 180,E1 17669.72,E2 17669.72} C_VEL
LIN {X 0,Y 263.692,Z 672.129,A -85,B 0,C 180,E1 17671.879,E2 17671.879} C_VEL
LIN {X 0,Y 257.984,Z 696.638,A -85,B 0,C 180,E1 17675.024,E2 17675.024} C_VEL
LIN {X 0,Y 251.368,Z 718.191,A -85,B 0,C 180,E1 17679.273,E2 17679.273} C_VEL
LIN {X 0,Y 245.255,Z 735.65,A -85,B 0,C 180,E1 17684.588,E2 17684.588} C_VEL
LIN {X 0,Y 240.5,Z 748.855,A -85,B 0,C 180,E1 17691.137,E2 17691.137} C_VEL
LIN {X 0,Y 237.92,Z 755.676,A -85,B 0,C 180,E1 17697.375,E2 17697.375} C_VEL
LIN {X 0,Y 236.486,Z 757.892,A -85,B 0,C 180,E1 17703.468,E2 17703.468} C_VEL
LIN {X 0,Y 236.923,Z 756.014,A -85,B 0,C 180,E1 17709.493,E2 17709.493} C_VEL
LIN {X 0,Y 238.919,Z 748.946,A -85,B 0,C 180,E1 17716.198,E2 17716.198} C_VEL
LIN {X 0,Y 242.548,Z 735.708,A -85,B 0,C 180,E1 17722.851,E2 17722.851} C_VEL
LIN {X 0,Y 247.377,Z 718.34,A -85,B 0,C 180,E1 17728.251,E2 17728.251} C_VEL
LIN {X 0,Y 253.127,Z 696.02,A -85,B 0,C 180,E1 17732.775,E2 17732.775} C_VEL
LIN {X 0,Y 258.185,Z 670.868,A -85,B 0,C 180,E1 17736.072,E2 17736.072} C_VEL
LIN {X 0,Y 262.045,Z 641.849,A -85,B 0,C 180,E1 17738.306,E2 17738.306} C_VEL
LIN {X 0,Y 264.032,Z 598.477,A -85,B 0,C 180,E1 17739.804,E2 17739.804} C_VEL
LIN {X 0,Y 252.573,Z 566.863,A -85,B 0,C 180,E1 17742.532,E2 17742.532} C_VEL
LIN {X 0,Y 236.541,Z 534.509,A -85,B 0,C 180,E1 17746.465,E2 17746.465} C_VEL
LIN {X 0,Y 234.815,Z 529.66,A -85,B 0,C 180,E1 17747.058,E2 17747.058} C_VEL
LIN {X 0,Y 234.13,Z 529.66,A -85,B 0,C 180,E1 17756.816,E2 17756.816} C_VEL
LIN {X 0,Y 233.736,Z 529.66,A -85,B 0,C 180,E1 17765.522,E2 17765.522} C_VEL
LIN {X 0,Y 233.698,Z 530.047,A -85,B 0,C 180,E1 17767.39,E2 17767.39} C_VEL
LIN {X 0,Y 253.81,Z 576.205,A -85,B 0,C 180,E1 17773.572,E2 17773.572} C_VEL
LIN {X 0,Y 265.35,Z 610.134,A -85,B 0,C 180,E1 17778.115,E2 17778.115} C_VEL
LIN {X 0,Y 267.771,Z 621.339,A -85,B 0,C 180,E1 17779.632,E2 17779.632} C_VEL
LIN {X 0,Y 259.84,Z 656.469,A -85,B 0,C 180,E1 17783.722,E2 17783.722} C_VEL
LIN {X 0,Y 251.928,Z 686.597,A -85,B 0,C 180,E1 17788.889,E2 17788.889} C_VEL
LIN {X 0,Y 245.266,Z 711.354,A -85,B 0,C 180,E1 17794.972,E2 17794.972} C_VEL
LIN {X 0,Y 240.313,Z 731.612,A -85,B 0,C 180,E1 17802.17,E2 17802.17} C_VEL
LIN {X 0,Y 237.753,Z 746.047,A -85,B 0,C 180,E1 17810.005,E2 17810.005} C_VEL
LIN {X 0,Y 236.936,Z 753.255,A -85,B 0,C 180,E1 17816.344,E2 17816.344} C_VEL
LIN {X 0,Y 237.259,Z 757.201,A -85,B 0,C 180,E1 17823.642,E2 17823.642} C_VEL
LIN {X 0,Y 238.952,Z 756.891,A -85,B 0,C 180,E1 17830.916,E2 17830.916} C_VEL
LIN {X 0,Y 244.425,Z 750.965,A -85,B 0,C 180,E1 17839.844,E2 17839.844} C_VEL
LIN {X 0,Y 254.89,Z 739.034,A -85,B 0,C 180,E1 17848.264,E2 17848.264} C_VEL
LIN {X 0,Y 272.455,Z 719.933,A -85,B 0,C 180,E1 17856.309,E2 17856.309} C_VEL
LIN {X 0,Y 292.976,Z 699.062,A -85,B 0,C 180,E1 17862.028,E2 17862.028} C_VEL
LIN {X 0,Y 293.648,Z 698.526,A -85,B 0,C 180,E1 17862.624,E2 17862.624} C_VEL
LIN {X 0,Y 269.845,Z 726.724,A -85,B 0,C 180,E1 17869.29,E2 17869.29} C_VEL
LIN {X 0,Y 251.544,Z 751.655,A -85,B 0,C 180,E1 17878.34,E2 17878.34} C_VEL
LIN {X 0,Y 241.394,Z 768.38,A -85,B 0,C 180,E1 17887.973,E2 17887.973} C_VEL
LIN {X 0,Y 237.531,Z 777.481,A -85,B 0,C 180,E1 17897.155,E2 17897.155} C_VEL
LIN {X 0,Y 236.877,Z 780.114,A -85,B 0,C 180,E1 17902.682,E2 17902.682} C_VEL
LIN {X 0,Y 237.032,Z 780.805,A -85,B 0,C 180,E1 17910.002,E2 17910.002} C_VEL
LIN {X 0,Y 236.91,Z 780.366,A -85,B 0,C 180,E1 17913.653,E2 17913.653} C_VEL
LIN {X 0,Y 237.235,Z 776.088,A -85,B 0,C 180,E1 17919.882,E2 17919.882} C_VEL
LIN {X 0,Y 238.479,Z 766.329,A -85,B 0,C 180,E1 17926.545,E2 17926.545} C_VEL
LIN {X 0,Y 241.447,Z 750.762,A -85,B 0,C 180,E1 17932.994,E2 17932.994} C_VEL
LIN {X 0,Y 249.385,Z 720.126,A -85,B 0,C 180,E1 17942.11,E2 17942.11} C_VEL
LIN {X 0,Y 257.524,Z 691.567,A -85,B 0,C 180,E1 17947.998,E2 17947.998} C_VEL
LIN {X 0,Y 266.484,Z 657.96,A -85,B 0,C 180,E1 17952.807,E2 17952.807} C_VEL
LIN {X 0,Y 273.109,Z 627.785,A -85,B 0,C 180,E1 17955.829,E2 17955.829} C_VEL
LIN {X 0,Y 261.248,Z 592.67,A -85,B 0,C 180,E1 17960.471,E2 17960.471} C_VEL
LIN {X 0,Y 244.849,Z 554.037,A -85,B 0,C 180,E1 17965.398,E2 17965.398} C_VEL
LIN {X 0,Y 234.021,Z 529.66,A -85,B 0,C 180,E1 17968.952,E2 17968.952} C_VEL
LIN {X 0,Y 234.369,Z 529.66,A -85,B 0,C 180,E1 17977.28,E2 17977.28} C_VEL
LIN {X 0,Y 234.799,Z 529.66,A -85,B 0,C 180,E1 17984.03,E2 17984.03} C_VEL
LIN {X 0,Y 232.701,Z 529.66,A -85,B 0,C 180,E1 17987.193,E2 17987.193} C_VEL
LIN {X 0,Y 227.733,Z 529.66,A -85,B 0,C 180,E1 17992.574,E2 17992.574} C_VEL
LIN {X 0,Y 228.53,Z 529.66,A -85,B 0,C 180,E1 18000.005,E2 18000.005} C_VEL
LIN {X 0,Y 227.784,Z 529.66,A -85,B 0,C 180,E1 18007.619,E2 18007.619} C_VEL
LIN {X 0,Y 227.199,Z 529.768,A -85,B 0,C 180,E1 18013.08,E2 18013.08} C_VEL
LIN {X 0,Y 229.336,Z 535.125,A -85,B 0,C 180,E1 18014.29,E2 18014.29} C_VEL
LIN {X 0,Y 232.107,Z 539.004,A -85,B 0,C 180,E1 18015.592,E2 18015.592} C_VEL
LIN {X 0,Y 243.398,Z 557.257,A -85,B 0,C 180,E1 18020.252,E2 18020.252} C_VEL
LIN {X 0,Y 255.754,Z 582.277,A -85,B 0,C 180,E1 18024.524,E2 18024.524} C_VEL
LIN {X 0,Y 264.37,Z 606.237,A -85,B 0,C 180,E1 18027.288,E2 18027.288} C_VEL
LIN {X 0,Y 261.782,Z 645.461,A -85,B 0,C 180,E1 18028.716,E2 18028.716} C_VEL
LIN {X 0,Y 257.094,Z 673.855,A -85,B 0,C 180,E1 18030.964,E2 18030.964} C_VEL
LIN {X 0,Y 250.504,Z 700.204,A -85,B 0,C 180,E1 18034.557,E2 18034.557} C_VEL
LIN {X 0,Y 243.339,Z 721.839,A -85,B 0,C 180,E1 18039.208,E2 18039.208} C_VEL
LIN {X 0,Y 237.019,Z 738.633,A -85,B 0,C 180,E1 18044.883,E2 18044.883} C_VEL
LIN {X 0,Y 232.599,Z 750.04,A -85,B 0,C 180,E1 18051.131,E2 18051.131} C_VEL
LIN {X 0,Y 229.577,Z 757.086,A -85,B 0,C 180,E1 18058.711,E2 18058.711} C_VEL
LIN {X 0,Y 228.685,Z 758.229,A -85,B 0,C 180,E1 18062.488,E2 18062.488} C_VEL
LIN {X 0,Y 228.683,Z 757.48,A -85,B 0,C 180,E1 18067.501,E2 18067.501} C_VEL
LIN {X 0,Y 230.49,Z 751.533,A -85,B 0,C 180,E1 18074.817,E2 18074.817} C_VEL
LIN {X 0,Y 233.776,Z 740.044,A -85,B 0,C 180,E1 18081.648,E2 18081.648} C_VEL
LIN {X 0,Y 238.806,Z 722.973,A -85,B 0,C 180,E1 18087.735,E2 18087.735} C_VEL
LIN {X 0,Y 244.743,Z 701.281,A -85,B 0,C 180,E1 18092.689,E2 18092.689} C_VEL
LIN {X 0,Y 250.492,Z 675.313,A -85,B 0,C 180,E1 18096.458,E2 18096.458} C_VEL
LIN {X 0,Y 254.726,Z 647.049,A -85,B 0,C 180,E1 18098.911,E2 18098.911} C_VEL
LIN {X 0,Y 257.019,Z 614.119,A -85,B 0,C 180,E1 18100.25,E2 18100.25} C_VEL
LIN {X 0,Y 256.776,Z 598.361,A -85,B 0,C 180,E1 18100.819,E2 18100.819} C_VEL
LIN {X 0,Y 244.02,Z 564.588,A -85,B 0,C 180,E1 18103.993,E2 18103.993} C_VEL
LIN {X 0,Y 226.907,Z 530.916,A -85,B 0,C 180,E1 18108.508,E2 18108.508} C_VEL
LIN {X 0,Y 226.806,Z 529.66,A -85,B 0,C 180,E1 18108.591,E2 18108.591} C_VEL
LIN {X 0,Y 226.039,Z 529.66,A -85,B 0,C 180,E1 18117.858,E2 18117.858} C_VEL
LIN {X 0,Y 225.838,Z 530.253,A -85,B 0,C 180,E1 18125.946,E2 18125.946} C_VEL
LIN {X 0,Y 246.108,Z 576.606,A -85,B 0,C 180,E1 18132.502,E2 18132.502} C_VEL
LIN {X 0,Y 257.733,Z 610.72,A -85,B 0,C 180,E1 18137.27,E2 18137.27} C_VEL
LIN {X 0,Y 260.525,Z 622.653,A -85,B 0,C 180,E1 18138.972,E2 18138.972} C_VEL
LIN {X 0,Y 252.564,Z 656.589,A -85,B 0,C 180,E1 18143.039,E2 18143.039} C_VEL
LIN {X 0,Y 244.401,Z 686.786,A -85,B 0,C 180,E1 18148.339,E2 18148.339} C_VEL
LIN {X 0,Y 237.523,Z 711.604,A -85,B 0,C 180,E1 18154.602,E2 18154.602} C_VEL
LIN {X 0,Y 232.433,Z 731.931,A -85,B 0,C 180,E1 18162.034,E2 18162.034} C_VEL
LIN {X 0,Y 229.879,Z 746.152,A -85,B 0,C 180,E1 18169.936,E2 18169.936} C_VEL
LIN {X 0,Y 228.996,Z 754.818,A -85,B 0,C 180,E1 18178.107,E2 18178.107} C_VEL
LIN {X 0,Y 229.375,Z 757.614,A -85,B 0,C 180,E1 18183.767,E2 18183.767} C_VEL
LIN {X 0,Y 231.544,Z 757.429,A -85,B 0,C 180,E1 18192.167,E2 18192.167} C_VEL
LIN {X 0,Y 237.092,Z 752.348,A -85,B 0,C 180,E1 18200.485,E2 18200.485} C_VEL
LIN {X 0,Y 248.256,Z 741.256,A -85,B 0,C 180,E1 18209.09,E2 18209.09} C_VEL
LIN {X 0,Y 267.405,Z 722.862,A -85,B 0,C 180,E1 18217.435,E2 18217.435} C_VEL
LIN {X 0,Y 284.979,Z 706.966,A -85,B 0,C 180,E1 18222.222,E2 18222.222} C_VEL
LIN {X 0,Y 256.419,Z 738.298,A -85,B 0,C 180,E1 18231.3,E2 18231.3} C_VEL
LIN {X 0,Y 241.21,Z 757.671,A -85,B 0,C 180,E1 18239.97,E2 18239.97} C_VEL
LIN {X 0,Y 232.719,Z 770.807,A -85,B 0,C 180,E1 18249.108,E2 18249.108} C_VEL
LIN {X 0,Y 229.348,Z 778.334,A -85,B 0,C 180,E1 18258.618,E2 18258.618} C_VEL
LIN {X 0,Y 228.892,Z 780.06,A -85,B 0,C 180,E1 18266.222,E2 18266.222} C_VEL
LIN {X 0,Y 228.999,Z 780.008,A -85,B 0,C 180,E1 18273.78,E2 18273.78} C_VEL
LIN {X 0,Y 229.371,Z 776.006,A -85,B 0,C 180,E1 18280.035,E2 18280.035} C_VEL
LIN {X 0,Y 230.771,Z 766.146,A -85,B 0,C 180,E1 18287.114,E2 18287.114} C_VEL
LIN {X 0,Y 233.972,Z 750.876,A -85,B 0,C 180,E1 18293.711,E2 18293.711} C_VEL
LIN {X 0,Y 243.346,Z 714.273,A -85,B 0,C 180,E1 18303.926,E2 18303.926} C_VEL
LIN {X 0,Y 252.362,Z 683.575,A -85,B 0,C 180,E1 18309.925,E2 18309.925} C_VEL
LIN {X 0,Y 261.536,Z 649.134,A -85,B 0,C 180,E1 18314.52,E2 18314.52} C_VEL
LIN {X 0,Y 265.693,Z 629.36,A -85,B 0,C 180,E1 18316.485,E2 18316.485} C_VEL
LIN {X 0,Y 254.068,Z 594.564,A -85,B 0,C 180,E1 18321.289,E2 18321.289} C_VEL
LIN {X 0,Y 238.586,Z 557.537,A -85,B 0,C 180,E1 18326.215,E2 18326.215} C_VEL
LIN {X 0,Y 226.037,Z 529.66,A -85,B 0,C 180,E1 18330.371,E2 18330.371} C_VEL
LIN {X 0,Y 226.479,Z 529.66,A -85,B 0,C 180,E1 18338.879,E2 18338.879} C_VEL
LIN {X 0,Y 227.298,Z 529.66,A -85,B 0,C 180,E1 18348.517,E2 18348.517} C_VEL
LIN {X 0,Y 227.733,Z 529.66,A -85,B 0,C 180,E1 18352.574,E2 18352.574} C_VEL
LIN {X 0,Y 225.558,Z 529.66,A -85,B 0,C 180,E1 18355.834,E2 18355.834} C_VEL
LIN {X 0,Y 220.363,Z 529.66,A -85,B 0,C 180,E1 18361.377,E2 18361.377} C_VEL
LIN {X 0,Y 219.608,Z 530.414,A -85,B 0,C 180,E1 18369.522,E2 18369.522} C_VEL
LIN {X 0,Y 222.059,Z 535.489,A -85,B 0,C 180,E1 18371.147,E2 18371.147} C_VEL
LIN {X 0,Y 224.483,Z 538.643,A -85,B 0,C 180,E1 18372.501,E2 18372.501} C_VEL
LIN {X 0,Y 235.666,Z 556.38,A -85,B 0,C 180,E1 18377.832,E2 18377.832} C_VEL
LIN {X 0,Y 247.892,Z 579.958,A -85,B 0,C 180,E1 18382.532,E2 18382.532} C_VEL
LIN {X 0,Y 257.999,Z 606.828,A -85,B 0,C 180,E1 18386.016,E2 18386.016} C_VEL
LIN {X 0,Y 258.262,Z 615.586,A -85,B 0,C 180,E1 18386.418,E2 18386.418} C_VEL
LIN {X 0,Y 255.608,Z 647.725,A -85,B 0,C 180,E1 18387.68,E2 18387.68} C_VEL
LIN {X 0,Y 250.561,Z 675.783,A -85,B 0,C 180,E1 18390.024,E2 18390.024} C_VEL
LIN {X 0,Y 243.67,Z 701.707,A -85,B 0,C 180,E1 18393.707,E2 18393.707} C_VEL
LIN {X 0,Y 236.304,Z 722.627,A -85,B 0,C 180,E1 18398.37,E2 18398.37} C_VEL
LIN {X 0,Y 230.003,Z 738.4,A -85,B 0,C 180,E1 18403.804,E2 18403.804} C_VEL
LIN {X 0,Y 225.059,Z 750.278,A -85,B 0,C 180,E1 18410.41,E2 18410.41} C_VEL
LIN {X 0,Y 222.176,Z 756.748,A -85,B 0,C 180,E1 18417.086,E2 18417.086} C_VEL
LIN {X 0,Y 220.791,Z 758.644,A -85,B 0,C 180,E1 18422.693,E2 18422.693} C_VEL
LIN {X 0,Y 221.201,Z 756.492,A -85,B 0,C 180,E1 18430.055,E2 18430.055} C_VEL
LIN {X 0,Y 223.519,Z 748.97,A -85,B 0,C 180,E1 18437.299,E2 18437.299} C_VEL
LIN {X 0,Y 227.557,Z 735.742,A -85,B 0,C 180,E1 18444.134,E2 18444.134} C_VEL
LIN {X 0,Y 233.103,Z 717.454,A -85,B 0,C 180,E1 18449.998,E2 18449.998} C_VEL
LIN {X 0,Y 239.398,Z 694.375,A -85,B 0,C 180,E1 18454.744,E2 18454.744} C_VEL
LIN {X 0,Y 245.073,Z 667.091,A -85,B 0,C 180,E1 18458.248,E2 18458.248} C_VEL
LIN {X 0,Y 248.99,Z 637.763,A -85,B 0,C 180,E1 18460.366,E2 18460.366} C_VEL
LIN {X 0,Y 250.416,Z 601.24,A -85,B 0,C 180,E1 18461.648,E2 18461.648} C_VEL
LIN {X 0,Y 238.206,Z 568.657,A -85,B 0,C 180,E1 18464.828,E2 18464.828} C_VEL
LIN {X 0,Y 220.902,Z 535.111,A -85,B 0,C 180,E1 18469.6,E2 18469.6} C_VEL
LIN {X 0,Y 218.606,Z 529.66,A -85,B 0,C 180,E1 18470.615,E2 18470.615} C_VEL
LIN {X 0,Y 218.06,Z 529.66,A -85,B 0,C 180,E1 18478.972,E2 18478.972} C_VEL
LIN {X 0,Y 217.899,Z 529.66,A -85,B 0,C 180,E1 18484.315,E2 18484.315} C_VEL
LIN {X 0,Y 238.545,Z 577.355,A -85,B 0,C 180,E1 18491.431,E2 18491.431} C_VEL
LIN {X 0,Y 250.088,Z 611.293,A -85,B 0,C 180,E1 18496.389,E2 18496.389} C_VEL
LIN {X 0,Y 253.134,Z 624.504,A -85,B 0,C 180,E1 18498.339,E2 18498.339} C_VEL
LIN {X 0,Y 244.78,Z 658.777,A -85,B 0,C 180,E1 18502.639,E2 18502.639} C_VEL
LIN {X 0,Y 236.316,Z 688.933,A -85,B 0,C 180,E1 18508.205,E2 18508.205} C_VEL
LIN {X 0,Y 229.392,Z 713.257,A -85,B 0,C 180,E1 18514.68,E2 18514.68} C_VEL
LIN {X 0,Y 224.316,Z 733.246,A -85,B 0,C 180,E1 18522.374,E2 18522.374} C_VEL
LIN {X 0,Y 221.785,Z 747.591,A -85,B 0,C 180,E1 18530.872,E2 18530.872} C_VEL
LIN {X 0,Y 221.114,Z 754.862,A -85,B 0,C 180,E1 18538.039,E2 18538.039} C_VEL
LIN {X 0,Y 221.511,Z 757.999,A -85,B 0,C 180,E1 18543.901,E2 18543.901} C_VEL
LIN {X 0,Y 223.497,Z 758.488,A -85,B 0,C 180,E1 18551.681,E2 18551.681} C_VEL
LIN {X 0,Y 229.792,Z 753.727,A -85,B 0,C 180,E1 18561.167,E2 18561.167} C_VEL
LIN {X 0,Y 243.226,Z 742.2,A -85,B 0,C 180,E1 18570.78,E2 18570.78} C_VEL
LIN {X 0,Y 263.775,Z 724.883,A -85,B 0,C 180,E1 18578.991,E2 18578.991} C_VEL
LIN {X 0,Y 274.761,Z 716.009,A -85,B 0,C 180,E1 18581.947,E2 18581.947} C_VEL
LIN {X 0,Y 275.316,Z 715.698,A -85,B 0,C 180,E1 18582.499,E2 18582.499} C_VEL
LIN {X 0,Y 251.429,Z 739.221,A -85,B 0,C 180,E1 18589.823,E2 18589.823} C_VEL
LIN {X 0,Y 234.36,Z 758.57,A -85,B 0,C 180,E1 18598.998,E2 18598.998} C_VEL
LIN {X 0,Y 225.212,Z 770.969,A -85,B 0,C 180,E1 18608.378,E2 18608.378} C_VEL
LIN {X 0,Y 221.503,Z 778.005,A -85,B 0,C 180,E1 18618.209,E2 18618.209} C_VEL
LIN {X 0,Y 221.007,Z 779.502,A -85,B 0,C 180,E1 18626.087,E2 18626.087} C_VEL
LIN {X 0,Y 221.24,Z 780.014,A -85,B 0,C 180,E1 18630.002,E2 18630.002} C_VEL
LIN {X 0,Y 221.088,Z 779.649,A -85,B 0,C 180,E1 18633.915,E2 18633.915} C_VEL
LIN {X 0,Y 221.529,Z 775.49,A -85,B 0,C 180,E1 18640.636,E2 18640.636} C_VEL
LIN {X 0,Y 223.334,Z 764.83,A -85,B 0,C 180,E1 18648.364,E2 18648.364} C_VEL
LIN {X 0,Y 227.145,Z 748.735,A -85,B 0,C 180,E1 18655.292,E2 18655.292} C_VEL
LIN {X 0,Y 232.151,Z 727.123,A -85,B 0,C 180,E1 18661.334,E2 18661.334} C_VEL
LIN {X 0,Y 242.833,Z 690.618,A -85,B 0,C 180,E1 18669.328,E2 18669.328} C_VEL
LIN {X 0,Y 252.213,Z 657.415,A -85,B 0,C 180,E1 18674.301,E2 18674.301} C_VEL
LIN {X 0,Y 258.404,Z 631.482,A -85,B 0,C 180,E1 18677.064,E2 18677.064} C_VEL
LIN {X 0,Y 247.056,Z 596.77,A -85,B 0,C 180,E1 18682.083,E2 18682.083} C_VEL
LIN {X 0,Y 231.758,Z 559.927,A -85,B 0,C 180,E1 18687.222,E2 18687.222} C_VEL
LIN {X 0,Y 218.203,Z 529.66,A -85,B 0,C 180,E1 18692.055,E2 18692.055} C_VEL
LIN {X 0,Y 218.646,Z 529.66,A -85,B 0,C 180,E1 18699.819,E2 18699.819} C_VEL
LIN {X 0,Y 219.305,Z 529.66,A -85,B 0,C 180,E1 18708.093,E2 18708.093} C_VEL
LIN {X 0,Y 220.237,Z 529.66,A -85,B 0,C 180,E1 18716.077,E2 18716.077} C_VEL
LIN {X 0,Y 220.363,Z 529.66,A -85,B 0,C 180,E1 18721.377,E2 18721.377} C_VEL
LIN {X 0,Y 217.679,Z 531.124,A -85,B 0,C 180,E1 18723.621,E2 18723.621} C_VEL
LIN {X 0,Y 214.25,Z 535.145,A -85,B 0,C 180,E1 18726.686,E2 18726.686} C_VEL
LIN {X 0,Y 214.763,Z 535.722,A -85,B 0,C 180,E1 18727.231,E2 18727.231} C_VEL
LIN {X 0,Y 217.037,Z 538.237,A -85,B 0,C 180,E1 18728.753,E2 18728.753} C_VEL
LIN {X 0,Y 225.935,Z 552.15,A -85,B 0,C 180,E1 18733.994,E2 18733.994} C_VEL
LIN {X 0,Y 236.655,Z 570.939,A -85,B 0,C 180,E1 18738.922,E2 18738.922} C_VEL
LIN {X 0,Y 247.415,Z 594.87,A -85,B 0,C 180,E1 18743.08,E2 18743.08} C_VEL
LIN {X 0,Y 252.793,Z 611.792,A -85,B 0,C 180,E1 18745.085,E2 18745.085} C_VEL
LIN {X 0,Y 249.8,Z 647.688,A -85,B 0,C 180,E1 18746.455,E2 18746.455} C_VEL
LIN {X 0,Y 244.481,Z 676.18,A -85,B 0,C 180,E1 18748.855,E2 18748.855} C_VEL
LIN {X 0,Y 237.415,Z 701.608,A -85,B 0,C 180,E1 18752.51,E2 18752.51} C_VEL
LIN {X 0,Y 229.61,Z 722.683,A -85,B 0,C 180,E1 18757.259,E2 18757.259} C_VEL
LIN {X 0,Y 222.518,Z 739.417,A -85,B 0,C 180,E1 18763.219,E2 18763.219} C_VEL
LIN {X 0,Y 217.526,Z 750.666,A -85,B 0,C 180,E1 18769.744,E2 18769.744} C_VEL
LIN {X 0,Y 214.731,Z 756.597,A -85,B 0,C 180,E1 18775.791,E2 18775.791} C_VEL
LIN {X 0,Y 213.254,Z 758.696,A -85,B 0,C 180,E1 18780.307,E2 18780.307} C_VEL
LIN {X 0,Y 212.819,Z 758.358,A -85,B 0,C 180,E1 18787.197,E2 18787.197} C_VEL
LIN {X 0,Y 214.624,Z 752.956,A -85,B 0,C 180,E1 18794.711,E2 18794.711} C_VEL
LIN {X 0,Y 218.094,Z 741.876,A -85,B 0,C 180,E1 18802.044,E2 18802.044} C_VEL
LIN {X 0,Y 223.438,Z 725.428,A -85,B 0,C 180,E1 18808.547,E2 18808.547} C_VEL
LIN {X 0,Y 229.711,Z 704.652,A -85,B 0,C 180,E1 18813.765,E2 18813.765} C_VEL
LIN {X 0,Y 235.914,Z 679.764,A -85,B 0,C 180,E1 18817.776,E2 18817.776} C_VEL
LIN {X 0,Y 240.745,Z 651.603,A -85,B 0,C 180,E1 18820.534,E2 18820.534} C_VEL
LIN {X 0,Y 243.453,Z 621.288,A -85,B 0,C 180,E1 18821.995,E2 18821.995} C_VEL
LIN {X 0,Y 243.632,Z 602.362,A -85,B 0,C 180,E1 18822.659,E2 18822.659} C_VEL
LIN {X 0,Y 230.814,Z 569.078,A -85,B 0,C 180,E1 18826.155,E2 18826.155} C_VEL
LIN {X 0,Y 215.168,Z 539.344,A -85,B 0,C 180,E1 18830.703,E2 18830.703} C_VEL
LIN {X 0,Y 210.514,Z 529.66,A -85,B 0,C 180,E1 18832.433,E2 18832.433} C_VEL
LIN {X 0,Y 209.93,Z 529.66,A -85,B 0,C 180,E1 18842.64,E2 18842.64} C_VEL
LIN {X 0,Y 230.789,Z 577.355,A -85,B 0,C 180,E1 18850.213,E2 18850.213} C_VEL
LIN {X 0,Y 242.553,Z 612.186,A -85,B 0,C 180,E1 18855.522,E2 18855.522} C_VEL
LIN {X 0,Y 245.73,Z 626.274,A -85,B 0,C 180,E1 18857.691,E2 18857.691} C_VEL
LIN {X 0,Y 237.115,Z 660.271,A -85,B 0,C 180,E1 18862.126,E2 18862.126} C_VEL
LIN {X 0,Y 228.27,Z 690.992,A -85,B 0,C 180,E1 18868.067,E2 18868.067} C_VEL
LIN {X 0,Y 220.835,Z 716.297,A -85,B 0,C 180,E1 18875.253,E2 18875.253} C_VEL
LIN {X 0,Y 216.197,Z 734.45,A -85,B 0,C 180,E1 18882.739,E2 18882.739} C_VEL
LIN {X 0,Y 213.798,Z 748.208,A -85,B 0,C 180,E1 18891.283,E2 18891.283} C_VEL
LIN {X 0,Y 213.345,Z 756.3,A -85,B 0,C 180,E1 18899.995,E2 18899.995} C_VEL
LIN {X 0,Y 214.367,Z 759.252,A -85,B 0,C 180,E1 18908.088,E2 18908.088} C_VEL
LIN {X 0,Y 217.819,Z 758.283,A -85,B 0,C 180,E1 18916.082,E2 18916.082} C_VEL
LIN {X 0,Y 228.038,Z 751.142,A -85,B 0,C 180,E1 18926.494,E2 18926.494} C_VEL
LIN {X 0,Y 247.656,Z 736.496,A -85,B 0,C 180,E1 18936.441,E2 18936.441} C_VEL
LIN {X 0,Y 264.723,Z 723.99,A -85,B 0,C 180,E1 18941.713,E2 18941.713} C_VEL
LIN {X 0,Y 265.922,Z 723.265,A -85,B 0,C 180,E1 18942.467,E2 18942.467} C_VEL
LIN {X 0,Y 241.819,Z 744.933,A -85,B 0,C 180,E1 18950.239,E2 18950.239} C_VEL
LIN {X 0,Y 225.178,Z 762.174,A -85,B 0,C 180,E1 18959.832,E2 18959.832} C_VEL
LIN {X 0,Y 216.503,Z 772.898,A -85,B 0,C 180,E1 18969.607,E2 18969.607} C_VEL
LIN {X 0,Y 213.67,Z 777.689,A -85,B 0,C 180,E1 18977.77,E2 18977.77} C_VEL
LIN {X 0,Y 213.116,Z 778.859,A -85,B 0,C 180,E1 18985.941,E2 18985.941} C_VEL
LIN {X 0,Y 213.341,Z 779.617,A -85,B 0,C 180,E1 18990.002,E2 18990.002} C_VEL
LIN {X 0,Y 213.177,Z 779.294,A -85,B 0,C 180,E1 18994.061,E2 18994.061} C_VEL
LIN {X 0,Y 213.582,Z 775.955,A -85,B 0,C 180,E1 19000.175,E2 19000.175} C_VEL
LIN {X 0,Y 215.249,Z 766.547,A -85,B 0,C 180,E1 19007.952,E2 19007.952} C_VEL
LIN {X 0,Y 219.113,Z 751.483,A -85,B 0,C 180,E1 19015.17,E2 19015.17} C_VEL
LIN {X 0,Y 224.336,Z 731.404,A -85,B 0,C 180,E1 19021.422,E2 19021.422} C_VEL
LIN {X 0,Y 238.806,Z 679.463,A -85,B 0,C 180,E1 19031.871,E2 19031.871} C_VEL
LIN {X 0,Y 248.364,Z 644.882,A -85,B 0,C 180,E1 19036.504,E2 19036.504} C_VEL
LIN {X 0,Y 250.948,Z 632.865,A -85,B 0,C 180,E1 19037.767,E2 19037.767} C_VEL
LIN {X 0,Y 240.21,Z 599.547,A -85,B 0,C 180,E1 19042.804,E2 19042.804} C_VEL
LIN {X 0,Y 225.862,Z 564.233,A -85,B 0,C 180,E1 19047.98,E2 19047.98} C_VEL
LIN {X 0,Y 210.269,Z 529.66,A -85,B 0,C 180,E1 19053.755,E2 19053.755} C_VEL
LIN {X 0,Y 210.952,Z 529.66,A -85,B 0,C 180,E1 19063.38,E2 19063.38} C_VEL
LIN {X 0,Y 211.774,Z 529.66,A -85,B 0,C 180,E1 19071.813,E2 19071.813} C_VEL
LIN {X 0,Y 212.703,Z 529.66,A -85,B 0,C 180,E1 19080.005,E2 19080.005} C_VEL
LIN {X 0,Y 212.167,Z 530.432,A -85,B 0,C 180,E1 19085,E2 19085} C_VEL
LIN {X 0,Y 214.382,Z 535.375,A -85,B 0,C 180,E1 19086.971,E2 19086.971} C_VEL
LIN {X 0,Y 214.763,Z 535.722,A -85,B 0,C 180,E1 19087.231,E2 19087.231} C_VEL
LIN {X 0,Y 217.915,Z 541.418,A -85,B 0,C 180,E1 19089.485,E2 19089.485} C_VEL
LIN {X 0,Y 223.189,Z 559.278,A -85,B 0,C 180,E1 19093.314,E2 19093.314} C_VEL
LIN {X 0,Y 223.609,Z 559.902,A -85,B 0,C 180,E1 19093.532,E2 19093.532} C_VEL
LIN {X 0,Y 234.37,Z 579.756,A -85,B 0,C 180,E1 19098.663,E2 19098.663} C_VEL
LIN {X 0,Y 244.229,Z 604.004,A -85,B 0,C 180,E1 19102.686,E2 19102.686} C_VEL
LIN {X 0,Y 247.115,Z 613.062,A -85,B 0,C 180,E1 19103.809,E2 19103.809} C_VEL
LIN {X 0,Y 244.174,Z 647.651,A -85,B 0,C 180,E1 19105.163,E2 19105.163} C_VEL
LIN {X 0,Y 238.771,Z 675.785,A -85,B 0,C 180,E1 19107.538,E2 19107.538} C_VEL
LIN {X 0,Y 231.223,Z 701.728,A -85,B 0,C 180,E1 19111.29,E2 19111.29} C_VEL
LIN {X 0,Y 222.958,Z 722.982,A -85,B 0,C 180,E1 19116.147,E2 19116.147} C_VEL
LIN {X 0,Y 215.27,Z 740.051,A -85,B 0,C 180,E1 19122.408,E2 19122.408} C_VEL
LIN {X 0,Y 209.665,Z 751.801,A -85,B 0,C 180,E1 19129.626,E2 19129.626} C_VEL
LIN {X 0,Y 206.521,Z 757.698,A -85,B 0,C 180,E1 19136.495,E2 19136.495} C_VEL
LIN {X 0,Y 204.87,Z 759.428,A -85,B 0,C 180,E1 19143.771,E2 19143.771} C_VEL
LIN {X 0,Y 205.96,Z 755.787,A -85,B 0,C 180,E1 19152.278,E2 19152.278} C_VEL
LIN {X 0,Y 208.817,Z 747.04,A -85,B 0,C 180,E1 19159.805,E2 19159.805} C_VEL
LIN {X 0,Y 213.781,Z 732.315,A -85,B 0,C 180,E1 19166.964,E2 19166.964} C_VEL
LIN {X 0,Y 220.372,Z 712.134,A -85,B 0,C 180,E1 19173.055,E2 19173.055} C_VEL
LIN {X 0,Y 227.074,Z 688.042,A -85,B 0,C 180,E1 19177.636,E2 19177.636} C_VEL
LIN {X 0,Y 232.804,Z 660.289,A -85,B 0,C 180,E1 19180.879,E2 19180.879} C_VEL
LIN {X 0,Y 236.282,Z 630.802,A -85,B 0,C 180,E1 19182.725,E2 19182.725} C_VEL
LIN {X 0,Y 237.189,Z 604.623,A -85,B 0,C 180,E1 19183.628,E2 19183.628} C_VEL
LIN {X 0,Y 224.243,Z 571.188,A -85,B 0,C 180,E1 19187.341,E2 19187.341} C_VEL
LIN {X 0,Y 207.984,Z 540.482,A -85,B 0,C 180,E1 19192.38,E2 19192.38} C_VEL
LIN {X 0,Y 202.483,Z 530.443,A -85,B 0,C 180,E1 19194.325,E2 19194.325} C_VEL
LIN {X 0,Y 202.041,Z 529.66,A -85,B 0,C 180,E1 19200.893,E2 19200.893} C_VEL
LIN {X 0,Y 223.241,Z 577.842,A -85,B 0,C 180,E1 19209.009,E2 19209.009} C_VEL
LIN {X 0,Y 235.044,Z 613.056,A -85,B 0,C 180,E1 19214.62,E2 19214.62} C_VEL
LIN {X 0,Y 238.573,Z 626.894,A -85,B 0,C 180,E1 19216.898,E2 19216.898} C_VEL
LIN {X 0,Y 229.694,Z 660.832,A -85,B 0,C 180,E1 19221.452,E2 19221.452} C_VEL
LIN {X 0,Y 220.602,Z 691.496,A -85,B 0,C 180,E1 19227.575,E2 19227.575} C_VEL
LIN {X 0,Y 213.11,Z 716.341,A -85,B 0,C 180,E1 19234.853,E2 19234.853} C_VEL
LIN {X 0,Y 208.061,Z 735.601,A -85,B 0,C 180,E1 19243.13,E2 19243.13} C_VEL
LIN {X 0,Y 205.865,Z 748.595,A -85,B 0,C 180,E1 19251.564,E2 19251.564} C_VEL
LIN {X 0,Y 205.443,Z 756.388,A -85,B 0,C 180,E1 19259.994,E2 19259.994} C_VEL
LIN {X 0,Y 206.563,Z 759.748,A -85,B 0,C 180,E1 19268.395,E2 19268.395} C_VEL
LIN {X 0,Y 210.262,Z 759.21,A -85,B 0,C 180,E1 19276.677,E2 19276.677} C_VEL
LIN {X 0,Y 220.392,Z 753.4,A -85,B 0,C 180,E1 19286.837,E2 19286.837} C_VEL
LIN {X 0,Y 239.75,Z 740.869,A -85,B 0,C 180,E1 19296.715,E2 19296.715} C_VEL
LIN {X 0,Y 256.43,Z 730.07,A -85,B 0,C 180,E1 19301.936,E2 19301.936} C_VEL
LIN {X 0,Y 254.244,Z 731.887,A -85,B 0,C 180,E1 19302.983,E2 19302.983} C_VEL
LIN {X 0,Y 226.875,Z 754.693,A -85,B 0,C 180,E1 19313.232,E2 19313.232} C_VEL
LIN {X 0,Y 211.901,Z 769.494,A -85,B 0,C 180,E1 19324.707,E2 19324.707} C_VEL
LIN {X 0,Y 206.993,Z 775.554,A -85,B 0,C 180,E1 19333.048,E2 19333.048} C_VEL
LIN {X 0,Y 205.327,Z 778.257,A -85,B 0,C 180,E1 19341.55,E2 19341.55} C_VEL
LIN {X 0,Y 205.441,Z 779.219,A -85,B 0,C 180,E1 19350.002,E2 19350.002} C_VEL
LIN {X 0,Y 205.286,Z 778.941,A -85,B 0,C 180,E1 19354.217,E2 19354.217} C_VEL
LIN {X 0,Y 205.716,Z 775.672,A -85,B 0,C 180,E1 19360.569,E2 19360.569} C_VEL
LIN {X 0,Y 207.429,Z 767.065,A -85,B 0,C 180,E1 19368.174,E2 19368.174} C_VEL
LIN {X 0,Y 211.308,Z 753.294,A -85,B 0,C 180,E1 19375.373,E2 19375.373} C_VEL
LIN {X 0,Y 217.024,Z 733.554,A -85,B 0,C 180,E1 19382.019,E2 19382.019} C_VEL
LIN {X 0,Y 223.163,Z 710.003,A -85,B 0,C 180,E1 19387.21,E2 19387.21} C_VEL
LIN {X 0,Y 228.973,Z 687.099,A -85,B 0,C 180,E1 19391.228,E2 19391.228} C_VEL
LIN {X 0,Y 239.044,Z 652.933,A -85,B 0,C 180,E1 19396.381,E2 19396.381} C_VEL
LIN {X 0,Y 243.434,Z 634.084,A -85,B 0,C 180,E1 19398.521,E2 19398.521} C_VEL
LIN {X 0,Y 232.858,Z 600.954,A -85,B 0,C 180,E1 19403.755,E2 19403.755} C_VEL
LIN {X 0,Y 218.519,Z 565.346,A -85,B 0,C 180,E1 19409.247,E2 19409.247} C_VEL
LIN {X 0,Y 206.675,Z 539.148,A -85,B 0,C 180,E1 19413.917,E2 19413.917} C_VEL
LIN {X 0,Y 205.874,Z 536.231,A -85,B 0,C 180,E1 19415.08,E2 19415.08} C_VEL
LIN {X 0,Y 202.794,Z 531.044,A -85,B 0,C 180,E1 19420.018,E2 19420.018} C_VEL
LIN {X 0,Y 202.726,Z 529.66,A -85,B 0,C 180,E1 19421.001,E2 19421.001} C_VEL
LIN {X 0,Y 203.335,Z 529.66,A -85,B 0,C 180,E1 19427.142,E2 19427.142} C_VEL
LIN {X 0,Y 204.408,Z 529.66,A -85,B 0,C 180,E1 19437.361,E2 19437.361} C_VEL
LIN {X 0,Y 208.247,Z 536.403,A -85,B 0,C 180,E1 19442.601,E2 19442.601} C_VEL
LIN {X 0,Y 209.92,Z 538.044,A -85,B 0,C 180,E1 19444.128,E2 19444.128} C_VEL
LIN {X 0,Y 213.87,Z 543.919,A -85,B 0,C 180,E1 19447.411,E2 19447.411} C_VEL
LIN {X 0,Y 223.609,Z 559.902,A -85,B 0,C 180,E1 19453.532,E2 19453.532} C_VEL
LIN {X 0,Y 227.245,Z 569.481,A -85,B 0,C 180,E1 19455.585,E2 19455.585} C_VEL
LIN {X 0,Y 231.878,Z 588.481,A -85,B 0,C 180,E1 19458.324,E2 19458.324} C_VEL
LIN {X 0,Y 240.992,Z 613.165,A -85,B 0,C 180,E1 19462.258,E2 19462.258} C_VEL
LIN {X 0,Y 241.407,Z 619.373,A -85,B 0,C 180,E1 19462.658,E2 19462.658} C_VEL
LIN {X 0,Y 238.26,Z 650.437,A -85,B 0,C 180,E1 19463.991,E2 19463.991} C_VEL
LIN {X 0,Y 232.201,Z 679.012,A -85,B 0,C 180,E1 19466.548,E2 19466.548} C_VEL
LIN {X 0,Y 224.252,Z 704.331,A -85,B 0,C 180,E1 19470.451,E2 19470.451} C_VEL
LIN {X 0,Y 215.506,Z 725.208,A -85,B 0,C 180,E1 19475.551,E2 19475.551} C_VEL
LIN {X 0,Y 207.794,Z 741.225,A -85,B 0,C 180,E1 19481.788,E2 19481.788} C_VEL
LIN {X 0,Y 202.617,Z 751.333,A -85,B 0,C 180,E1 19488.145,E2 19488.145} C_VEL
LIN {X 0,Y 199.186,Z 757.508,A -85,B 0,C 180,E1 19494.926,E2 19494.926} C_VEL
LIN {X 0,Y 197.081,Z 759.856,A -85,B 0,C 180,E1 19502.649,E2 19502.649} C_VEL
LIN {X 0,Y 197.45,Z 757.84,A -85,B 0,C 180,E1 19509.883,E2 19509.883} C_VEL
LIN {X 0,Y 199.579,Z 751.872,A -85,B 0,C 180,E1 19516.888,E2 19516.888} C_VEL
LIN {X 0,Y 203.873,Z 739.409,A -85,B 0,C 180,E1 19524.709,E2 19524.709} C_VEL
LIN {X 0,Y 209.895,Z 722.459,A -85,B 0,C 180,E1 19531.18,E2 19531.18} C_VEL
LIN {X 0,Y 216.891,Z 700.639,A -85,B 0,C 180,E1 19536.49,E2 19536.49} C_VEL
LIN {X 0,Y 223.492,Z 674.597,A -85,B 0,C 180,E1 19540.473,E2 19540.473} C_VEL
LIN {X 0,Y 228.309,Z 646.121,A -85,B 0,C 180,E1 19543.027,E2 19543.027} C_VEL
LIN {X 0,Y 230.961,Z 607.517,A -85,B 0,C 180,E1 19544.591,E2 19544.591} C_VEL
LIN {X 0,Y 218.232,Z 574.484,A -85,B 0,C 180,E1 19548.436,E2 19548.436} C_VEL
LIN {X 0,Y 203.09,Z 545.599,A -85,B 0,C 180,E1 19553.388,E2 19553.388} C_VEL
LIN {X 0,Y 194.395,Z 530.872,A -85,B 0,C 180,E1 19556.644,E2 19556.644} C_VEL
LIN {X 0,Y 194.25,Z 529.66,A -85,B 0,C 180,E1 19557.061,E2 19557.061} C_VEL
LIN {X 0,Y 194.136,Z 530.022,A -85,B 0,C 180,E1 19559.02,E2 19559.02} C_VEL
LIN {X 0,Y 215.164,Z 577.116,A -85,B 0,C 180,E1 19567.535,E2 19567.535} C_VEL
LIN {X 0,Y 227.052,Z 612.218,A -85,B 0,C 180,E1 19573.393,E2 19573.393} C_VEL
LIN {X 0,Y 230.988,Z 629.182,A -85,B 0,C 180,E1 19576.264,E2 19576.264} C_VEL
LIN {X 0,Y 221.436,Z 664.121,A -85,B 0,C 180,E1 19581.234,E2 19581.234} C_VEL
LIN {X 0,Y 212.146,Z 694.279,A -85,B 0,C 180,E1 19587.663,E2 19587.663} C_VEL
LIN {X 0,Y 204.588,Z 719.153,A -85,B 0,C 180,E1 19595.482,E2 19595.482} C_VEL
LIN {X 0,Y 199.949,Z 736.7,A -85,B 0,C 180,E1 19603.554,E2 19603.554} C_VEL
LIN {X 0,Y 197.826,Z 749.764,A -85,B 0,C 180,E1 19612.564,E2 19612.564} C_VEL
LIN {X 0,Y 197.54,Z 756.356,A -85,B 0,C 180,E1 19619.994,E2 19619.994} C_VEL
LIN {X 0,Y 199.023,Z 760.374,A -85,B 0,C 180,E1 19629.726,E2 19629.726} C_VEL
LIN {X 0,Y 206.114,Z 758.832,A -85,B 0,C 180,E1 19641.466,E2 19641.466} C_VEL
LIN {X 0,Y 218.95,Z 752.204,A -85,B 0,C 180,E1 19651.118,E2 19651.118} C_VEL
LIN {X 0,Y 240.558,Z 739.943,A -85,B 0,C 180,E1 19660.007,E2 19660.007} C_VEL
LIN {X 0,Y 247.668,Z 735.906,A -85,B 0,C 180,E1 19662.076,E2 19662.076} C_VEL
LIN {X 0,Y 218.962,Z 757.354,A -85,B 0,C 180,E1 19672.916,E2 19672.916} C_VEL
LIN {X 0,Y 204.675,Z 769.759,A -85,B 0,C 180,E1 19683.748,E2 19683.748} C_VEL
LIN {X 0,Y 199.302,Z 775.424,A -85,B 0,C 180,E1 19692.373,E2 19692.373} C_VEL
LIN {X 0,Y 197.459,Z 777.688,A -85,B 0,C 180,E1 19701.21,E2 19701.21} C_VEL
LIN {X 0,Y 197.365,Z 777.471,A -85,B 0,C 180,E1 19705.617,E2 19705.617} C_VEL
LIN {X 0,Y 197.54,Z 778.818,A -85,B 0,C 180,E1 19710.002,E2 19710.002} C_VEL
LIN {X 0,Y 197.334,Z 778.029,A -85,B 0,C 180,E1 19716.289,E2 19716.289} C_VEL
LIN {X 0,Y 198.41,Z 772.499,A -85,B 0,C 180,E1 19724.312,E2 19724.312} C_VEL
LIN {X 0,Y 201.235,Z 761.983,A -85,B 0,C 180,E1 19732.022,E2 19732.022} C_VEL
LIN {X 0,Y 206.58,Z 745.401,A -85,B 0,C 180,E1 19739.486,E2 19739.486} C_VEL
LIN {X 0,Y 213.269,Z 724.273,A -85,B 0,C 180,E1 19745.624,E2 19745.624} C_VEL
LIN {X 0,Y 219.546,Z 699.476,A -85,B 0,C 180,E1 19750.381,E2 19750.381} C_VEL
LIN {X 0,Y 224.562,Z 677.874,A -85,B 0,C 180,E1 19753.535,E2 19753.535} C_VEL
LIN {X 0,Y 234.653,Z 643.245,A -85,B 0,C 180,E1 19758.343,E2 19758.343} C_VEL
LIN {X 0,Y 235.963,Z 635.32,A -85,B 0,C 180,E1 19759.293,E2 19759.293} C_VEL
LIN {X 0,Y 225.055,Z 600.891,A -85,B 0,C 180,E1 19764.969,E2 19764.969} C_VEL
LIN {X 0,Y 210.836,Z 565.697,A -85,B 0,C 180,E1 19770.703,E2 19770.703} C_VEL
LIN {X 0,Y 205.698,Z 553.453,A -85,B 0,C 180,E1 19772.994,E2 19772.994} C_VEL
LIN {X 0,Y 204.147,Z 543.621,A -85,B 0,C 180,E1 19775.859,E2 19775.859} C_VEL
LIN {X 0,Y 201.306,Z 537.981,A -85,B 0,C 180,E1 19781.004,E2 19781.004} C_VEL
LIN {X 0,Y 201.01,Z 537.006,A -85,B 0,C 180,E1 19793.54,E2 19793.54} C_VEL
LIN {X 0,Y 203.058,Z 538.375,A -85,B 0,C 180,E1 19797.377,E2 19797.377} C_VEL
LIN {X 0,Y 208.151,Z 546.115,A -85,B 0,C 180,E1 19803.642,E2 19803.642} C_VEL
LIN {X 0,Y 213.508,Z 554.788,A -85,B 0,C 180,E1 19808.131,E2 19808.131} C_VEL
LIN {X 0,Y 222.559,Z 569.713,A -85,B 0,C 180,E1 19813.732,E2 19813.732} C_VEL
LIN {X 0,Y 231.878,Z 588.481,A -85,B 0,C 180,E1 19818.324,E2 19818.324} C_VEL
LIN {X 0,Y 233.188,Z 596.453,A -85,B 0,C 180,E1 19819.17,E2 19819.17} C_VEL
LIN {X 0,Y 233.799,Z 609.523,A -85,B 0,C 180,E1 19820.037,E2 19820.037} C_VEL
LIN {X 0,Y 234.168,Z 610.783,A -85,B 0,C 180,E1 19820.213,E2 19820.213} C_VEL
LIN {X 0,Y 236.22,Z 619.006,A -85,B 0,C 180,E1 19821.225,E2 19821.225} C_VEL
LIN {X 0,Y 232.828,Z 651.088,A -85,B 0,C 180,E1 19822.605,E2 19822.605} C_VEL
LIN {X 0,Y 226.541,Z 679.397,A -85,B 0,C 180,E1 19825.171,E2 19825.171} C_VEL
LIN {X 0,Y 218.207,Z 704.671,A -85,B 0,C 180,E1 19829.119,E2 19829.119} C_VEL
LIN {X 0,Y 208.955,Z 725.637,A -85,B 0,C 180,E1 19834.327,E2 19834.327} C_VEL
LIN {X 0,Y 200.359,Z 742.427,A -85,B 0,C 180,E1 19841.134,E2 19841.134} C_VEL
LIN {X 0,Y 194.191,Z 753.524,A -85,B 0,C 180,E1 19848.902,E2 19848.902} C_VEL
LIN {X 0,Y 190.71,Z 758.947,A -85,B 0,C 180,E1 19856.365,E2 19856.365} C_VEL
LIN {X 0,Y 189.34,Z 760.2,A -85,B 0,C 180,E1 19861.431,E2 19861.431} C_VEL
LIN {X 0,Y 189.351,Z 758.73,A -85,B 0,C 180,E1 19868.983,E2 19868.983} C_VEL
LIN {X 0,Y 191.418,Z 753.198,A -85,B 0,C 180,E1 19876.318,E2 19876.318} C_VEL
LIN {X 0,Y 195.665,Z 741.497,A -85,B 0,C 180,E1 19884.466,E2 19884.466} C_VEL
LIN {X 0,Y 202.206,Z 723.933,A -85,B 0,C 180,E1 19891.66,E2 19891.66} C_VEL
LIN {X 0,Y 209.573,Z 702.205,A -85,B 0,C 180,E1 19897.237,E2 19897.237} C_VEL
LIN {X 0,Y 216.619,Z 675.887,A -85,B 0,C 180,E1 19901.429,E2 19901.429} C_VEL
LIN {X 0,Y 221.532,Z 648.139,A -85,B 0,C 180,E1 19904.052,E2 19904.052} C_VEL
LIN {X 0,Y 224.34,Z 614.655,A -85,B 0,C 180,E1 19905.515,E2 19905.515} C_VEL
LIN {X 0,Y 223.536,Z 606.253,A -85,B 0,C 180,E1 19906.013,E2 19906.013} C_VEL
LIN {X 0,Y 210.345,Z 573.366,A -85,B 0,C 180,E1 19910.237,E2 19910.237} C_VEL
LIN {X 0,Y 195.228,Z 545.752,A -85,B 0,C 180,E1 19915.572,E2 19915.572} C_VEL
LIN {X 0,Y 188.93,Z 535.885,A -85,B 0,C 180,E1 19918.082,E2 19918.082} C_VEL
LIN {X 0,Y 207.74,Z 578.051,A -85,B 0,C 180,E1 19926.249,E2 19926.249} C_VEL
LIN {X 0,Y 219.133,Z 611.868,A -85,B 0,C 180,E1 19932.173,E2 19932.173} C_VEL
LIN {X 0,Y 223.747,Z 630.154,A -85,B 0,C 180,E1 19935.453,E2 19935.453} C_VEL
LIN {X 0,Y 213.906,Z 664.952,A -85,B 0,C 180,E1 19940.581,E2 19940.581} C_VEL
LIN {X 0,Y 204.589,Z 694.303,A -85,B 0,C 180,E1 19947.04,E2 19947.04} C_VEL
LIN {X 0,Y 196.829,Z 719.075,A -85,B 0,C 180,E1 19955.055,E2 19955.055} C_VEL
LIN {X 0,Y 191.858,Z 737.743,A -85,B 0,C 180,E1 19964.015,E2 19964.015} C_VEL
LIN {X 0,Y 189.872,Z 750.237,A -85,B 0,C 180,E1 19973.077,E2 19973.077} C_VEL
LIN {X 0,Y 189.709,Z 757.767,A -85,B 0,C 180,E1 19982.273,E2 19982.273} C_VEL
LIN {X 0,Y 192.639,Z 761.216,A -85,B 0,C 180,E1 19993.585,E2 19993.585} C_VEL
LIN {X 0,Y 198.836,Z 759.987,A -85,B 0,C 180,E1 20002.293,E2 20002.293} C_VEL
LIN {X 0,Y 216,Z 752.503,A -85,B 0,C 180,E1 20013.972,E2 20013.972} C_VEL
LIN {X 0,Y 237.366,Z 741.987,A -85,B 0,C 180,E1 20021.83,E2 20021.83} C_VEL
LIN {X 0,Y 233.404,Z 744.681,A -85,B 0,C 180,E1 20023.489,E2 20023.489} C_VEL
LIN {X 0,Y 207.787,Z 762.116,A -85,B 0,C 180,E1 20034.483,E2 20034.483} C_VEL
LIN {X 0,Y 194.016,Z 773.012,A -85,B 0,C 180,E1 20047.117,E2 20047.117} C_VEL
LIN {X 0,Y 190.207,Z 776.561,A -85,B 0,C 180,E1 20056.233,E2 20056.233} C_VEL
LIN {X 0,Y 189.472,Z 776.959,A -85,B 0,C 180,E1 20065.434,E2 20065.434} C_VEL
LIN {X 0,Y 189.656,Z 778.407,A -85,B 0,C 180,E1 20070.002,E2 20070.002} C_VEL
LIN {X 0,Y 189.468,Z 778.241,A -85,B 0,C 180,E1 20074.57,E2 20074.57} C_VEL
LIN {X 0,Y 190.043,Z 775.129,A -85,B 0,C 180,E1 20081.452,E2 20081.452} C_VEL
LIN {X 0,Y 192.369,Z 766.295,A -85,B 0,C 180,E1 20090.019,E2 20090.019} C_VEL
LIN {X 0,Y 197.281,Z 752.24,A -85,B 0,C 180,E1 20097.886,E2 20097.886} C_VEL
LIN {X 0,Y 204.232,Z 732.32,A -85,B 0,C 180,E1 20104.935,E2 20104.935} C_VEL
LIN {X 0,Y 211.408,Z 708.76,A -85,B 0,C 180,E1 20110.331,E2 20110.331} C_VEL
LIN {X 0,Y 217.493,Z 682.17,A -85,B 0,C 180,E1 20114.265,E2 20114.265} C_VEL
LIN {X 0,Y 220.679,Z 666.759,A -85,B 0,C 180,E1 20116.098,E2 20116.098} C_VEL
LIN {X 0,Y 228.784,Z 637.745,A -85,B 0,C 180,E1 20119.883,E2 20119.883} C_VEL
LIN {X 0,Y 218.161,Z 603.325,A -85,B 0,C 180,E1 20125.813,E2 20125.813} C_VEL
LIN {X 0,Y 204.66,Z 567.994,A -85,B 0,C 180,E1 20132.126,E2 20132.126} C_VEL
LIN {X 0,Y 202.273,Z 550.877,A -85,B 0,C 180,E1 20136.903,E2 20136.903} C_VEL
LIN {X 0,Y 199.732,Z 545.082,A -85,B 0,C 180,E1 20142.416,E2 20142.416} C_VEL
LIN {X 0,Y 201.49,Z 545.524,A -85,B 0,C 180,E1 20156.534,E2 20156.534} C_VEL
LIN {X 0,Y 206.436,Z 553.9,A -85,B 0,C 180,E1 20163.148,E2 20163.148} C_VEL
LIN {X 0,Y 213.195,Z 564.697,A -85,B 0,C 180,E1 20168.784,E2 20168.784} C_VEL
LIN {X 0,Y 223.243,Z 583.499,A -85,B 0,C 180,E1 20174.893,E2 20174.893} C_VEL
LIN {X 0,Y 232.724,Z 606.247,A -85,B 0,C 180,E1 20179.537,E2 20179.537} C_VEL
LIN {X 0,Y 234.168,Z 610.783,A -85,B 0,C 180,E1 20180.213,E2 20180.213} C_VEL
LIN {X 0,Y 234.269,Z 617.618,A -85,B 0,C 180,E1 20180.586,E2 20180.586} C_VEL
LIN {X 0,Y 229.951,Z 634.104,A -85,B 0,C 180,E1 20180.21,E2 20180.21} C_VEL
LIN {X 0,Y 225.405,Z 662.982,A -85,B 0,C 180,E1 20182.004,E2 20182.004} C_VEL
LIN {X 0,Y 217.766,Z 690.278,A -85,B 0,C 180,E1 20185.142,E2 20185.142} C_VEL
LIN {X 0,Y 208.429,Z 714.057,A -85,B 0,C 180,E1 20189.679,E2 20189.679} C_VEL
LIN {X 0,Y 198.542,Z 733.672,A -85,B 0,C 180,E1 20195.756,E2 20195.756} C_VEL
LIN {X 0,Y 190.041,Z 748.425,A -85,B 0,C 180,E1 20203.442,E2 20203.442} C_VEL
LIN {X 0,Y 184.406,Z 757.5,A -85,B 0,C 180,E1 20212.406,E2 20212.406} C_VEL
LIN {X 0,Y 181.658,Z 760.522,A -85,B 0,C 180,E1 20220.103,E2 20220.103} C_VEL
LIN {X 0,Y 181.164,Z 760.038,A -85,B 0,C 180,E1 20226.396,E2 20226.396} C_VEL
LIN {X 0,Y 183.27,Z 754.474,A -85,B 0,C 180,E1 20235.697,E2 20235.697} C_VEL
LIN {X 0,Y 187.482,Z 743.355,A -85,B 0,C 180,E1 20244.224,E2 20244.224} C_VEL
LIN {X 0,Y 193.98,Z 726.899,A -85,B 0,C 180,E1 20251.645,E2 20251.645} C_VEL
LIN {X 0,Y 201.499,Z 705.95,A -85,B 0,C 180,E1 20257.529,E2 20257.529} C_VEL
LIN {X 0,Y 208.883,Z 680.712,A -85,B 0,C 180,E1 20261.975,E2 20261.975} C_VEL
LIN {X 0,Y 214.481,Z 652.484,A -85,B 0,C 180,E1 20264.942,E2 20264.942} C_VEL
LIN {X 0,Y 217.674,Z 620.67,A -85,B 0,C 180,E1 20266.545,E2 20266.545} C_VEL
LIN {X 0,Y 217.67,Z 609.878,A -85,B 0,C 180,E1 20267.011,E2 20267.011} C_VEL
LIN {X 0,Y 204.999,Z 577.752,A -85,B 0,C 180,E1 20271.301,E2 20271.301} C_VEL
LIN {X 0,Y 190.487,Z 550.847,A -85,B 0,C 180,E1 20276.721,E2 20276.721} C_VEL
LIN {X 0,Y 187.754,Z 546.332,A -85,B 0,C 180,E1 20277.85,E2 20277.85} C_VEL
LIN {X 0,Y 186.172,Z 547.094,A -85,B 0,C 180,E1 20278.606,E2 20278.606} C_VEL
LIN {X 0,Y 201.717,Z 582.659,A -85,B 0,C 180,E1 20285.596,E2 20285.596} C_VEL
LIN {X 0,Y 212.573,Z 615.976,A -85,B 0,C 180,E1 20291.719,E2 20291.719} C_VEL
LIN {X 0,Y 216.373,Z 631.722,A -85,B 0,C 180,E1 20294.685,E2 20294.685} C_VEL
LIN {X 0,Y 206.422,Z 665.576,A -85,B 0,C 180,E1 20299.864,E2 20299.864} C_VEL
LIN {X 0,Y 196.523,Z 695.849,A -85,B 0,C 180,E1 20306.826,E2 20306.826} C_VEL
LIN {X 0,Y 188.666,Z 720.263,A -85,B 0,C 180,E1 20315.165,E2 20315.165} C_VEL
LIN {X 0,Y 183.767,Z 738.725,A -85,B 0,C 180,E1 20324.516,E2 20324.516} C_VEL
LIN {X 0,Y 181.968,Z 750.063,A -85,B 0,C 180,E1 20333.088,E2 20333.088} C_VEL
LIN {X 0,Y 181.817,Z 757.725,A -85,B 0,C 180,E1 20342.372,E2 20342.372} C_VEL
LIN {X 0,Y 183.121,Z 760.895,A -85,B 0,C 180,E1 20349.48,E2 20349.48} C_VEL
LIN {X 0,Y 187.724,Z 761.848,A -85,B 0,C 180,E1 20358.749,E2 20358.749} C_VEL
LIN {X 0,Y 202.559,Z 757.466,A -85,B 0,C 180,E1 20371.424,E2 20371.424} C_VEL
LIN {X 0,Y 227.179,Z 747.32,A -85,B 0,C 180,E1 20381.616,E2 20381.616} C_VEL
LIN {X 0,Y 228.282,Z 746.825,A -85,B 0,C 180,E1 20381.949,E2 20381.949} C_VEL
LIN {X 0,Y 199.753,Z 764.044,A -85,B 0,C 180,E1 20394.167,E2 20394.167} C_VEL
LIN {X 0,Y 186.604,Z 772.958,A -85,B 0,C 180,E1 20406.153,E2 20406.153} C_VEL
LIN {X 0,Y 182.414,Z 776.137,A -85,B 0,C 180,E1 20415.633,E2 20415.633} C_VEL
LIN {X 0,Y 181.565,Z 776.707,A -85,B 0,C 180,E1 20425.71,E2 20425.71} C_VEL
LIN {X 0,Y 181.755,Z 777.98,A -85,B 0,C 180,E1 20430.002,E2 20430.002} C_VEL
LIN {X 0,Y 181.589,Z 777.893,A -85,B 0,C 180,E1 20434.769,E2 20434.769} C_VEL
LIN {X 0,Y 182.212,Z 774.866,A -85,B 0,C 180,E1 20441.951,E2 20441.951} C_VEL
LIN {X 0,Y 184.973,Z 765.665,A -85,B 0,C 180,E1 20451.268,E2 20451.268} C_VEL
LIN {X 0,Y 190.885,Z 750.562,A -85,B 0,C 180,E1 20459.822,E2 20459.822} C_VEL
LIN {X 0,Y 198.437,Z 730.875,A -85,B 0,C 180,E1 20466.77,E2 20466.77} C_VEL
LIN {X 0,Y 206.235,Z 706.887,A -85,B 0,C 180,E1 20472.269,E2 20472.269} C_VEL
LIN {X 0,Y 212.714,Z 680.024,A -85,B 0,C 180,E1 20476.174,E2 20476.174} C_VEL
LIN {X 0,Y 217.431,Z 653.57,A -85,B 0,C 180,E1 20478.835,E2 20478.835} C_VEL
LIN {X 0,Y 221.388,Z 639.409,A -85,B 0,C 180,E1 20480.607,E2 20480.607} C_VEL
LIN {X 0,Y 210.768,Z 604.523,A -85,B 0,C 180,E1 20486.92,E2 20486.92} C_VEL
LIN {X 0,Y 204.021,Z 584.847,A -85,B 0,C 180,E1 20490.738,E2 20490.738} C_VEL
LIN {X 0,Y 200.661,Z 558.252,A -85,B 0,C 180,E1 20497.678,E2 20497.678} C_VEL
LIN {X 0,Y 198.356,Z 552.792,A -85,B 0,C 180,E1 20503.431,E2 20503.431} C_VEL
LIN {X 0,Y 200.099,Z 553.279,A -85,B 0,C 180,E1 20516.027,E2 20516.027} C_VEL
LIN {X 0,Y 204.642,Z 561.373,A -85,B 0,C 180,E1 20522.527,E2 20522.527} C_VEL
LIN {X 0,Y 211.08,Z 572.397,A -85,B 0,C 180,E1 20528.226,E2 20528.226} C_VEL
LIN {X 0,Y 219.984,Z 589.807,A -85,B 0,C 180,E1 20533.966,E2 20533.966} C_VEL
LIN {X 0,Y 228.642,Z 611.826,A -85,B 0,C 180,E1 20538.53,E2 20538.53} C_VEL
LIN {X 0,Y 231.088,Z 620.339,A -85,B 0,C 180,E1 20539.765,E2 20539.765} C_VEL
LIN {X 0,Y 229.951,Z 634.104,A -85,B 0,C 180,E1 20540.21,E2 20540.21} C_VEL
LIN {X 0,Y 225.188,Z 651.008,A -85,B 0,C 180,E1 20540.312,E2 20540.312} C_VEL
LIN {X 0,Y 219.889,Z 665.384,A -85,B 0,C 180,E1 20540.665,E2 20540.665} C_VEL
LIN {X 0,Y 219.352,Z 667.346,A -85,B 0,C 180,E1 20540.828,E2 20540.828} C_VEL
LIN {X 0,Y 211.226,Z 693.727,A -85,B 0,C 180,E1 20544.083,E2 20544.083} C_VEL
LIN {X 0,Y 201.337,Z 716.72,A -85,B 0,C 180,E1 20548.785,E2 20548.785} C_VEL
LIN {X 0,Y 191.317,Z 735.29,A -85,B 0,C 180,E1 20554.908,E2 20554.908} C_VEL
LIN {X 0,Y 183.097,Z 748.532,A -85,B 0,C 180,E1 20562.118,E2 20562.118} C_VEL
LIN {X 0,Y 176.893,Z 757.821,A -85,B 0,C 180,E1 20571.497,E2 20571.497} C_VEL
LIN {X 0,Y 173.709,Z 760.971,A -85,B 0,C 180,E1 20580.319,E2 20580.319} C_VEL
LIN {X 0,Y 173.634,Z 759.154,A -85,B 0,C 180,E1 20589.656,E2 20589.656} C_VEL
LIN {X 0,Y 176.333,Z 752.464,A -85,B 0,C 180,E1 20598.399,E2 20598.399} C_VEL
LIN {X 0,Y 181.36,Z 740.098,A -85,B 0,C 180,E1 20606.915,E2 20606.915} C_VEL
LIN {X 0,Y 188.475,Z 722.589,A -85,B 0,C 180,E1 20614.18,E2 20614.18} C_VEL
LIN {X 0,Y 196.523,Z 700.428,A -85,B 0,C 180,E1 20619.887,E2 20619.887} C_VEL
LIN {X 0,Y 203.675,Z 675.313,A -85,B 0,C 180,E1 20623.931,E2 20623.931} C_VEL
LIN {X 0,Y 209.064,Z 646.455,A -85,B 0,C 180,E1 20626.644,E2 20626.644} C_VEL
LIN {X 0,Y 211.477,Z 612.211,A -85,B 0,C 180,E1 20628.207,E2 20628.207} C_VEL
LIN {X 0,Y 199.237,Z 581.131,A -85,B 0,C 180,E1 20632.598,E2 20632.598} C_VEL
LIN {X 0,Y 186.213,Z 556.543,A -85,B 0,C 180,E1 20637.749,E2 20637.749} C_VEL
LIN {X 0,Y 183.171,Z 557.066,A -85,B 0,C 180,E1 20638.804,E2 20638.804} C_VEL
LIN {X 0,Y 197.17,Z 591.177,A -85,B 0,C 180,E1 20645.699,E2 20645.699} C_VEL
LIN {X 0,Y 207.075,Z 624.385,A -85,B 0,C 180,E1 20652.141,E2 20652.141} C_VEL
LIN {X 0,Y 208.676,Z 634.581,A -85,B 0,C 180,E1 20654.053,E2 20654.053} C_VEL
LIN {X 0,Y 198.138,Z 668.689,A -85,B 0,C 180,E1 20659.601,E2 20659.601} C_VEL
LIN {X 0,Y 188.21,Z 697.998,A -85,B 0,C 180,E1 20666.798,E2 20666.798} C_VEL
LIN {X 0,Y 180.48,Z 721.369,A -85,B 0,C 180,E1 20675.282,E2 20675.282} C_VEL
LIN {X 0,Y 175.653,Z 739.636,A -85,B 0,C 180,E1 20685.058,E2 20685.058} C_VEL
LIN {X 0,Y 173.892,Z 751.772,A -85,B 0,C 180,E1 20695.015,E2 20695.015} C_VEL
LIN {X 0,Y 174.223,Z 759.031,A -85,B 0,C 180,E1 20704.962,E2 20704.962} C_VEL
LIN {X 0,Y 177.281,Z 762.325,A -85,B 0,C 180,E1 20714.788,E2 20714.788} C_VEL
